REGION Network 61: PHMI Servo Enable CMs
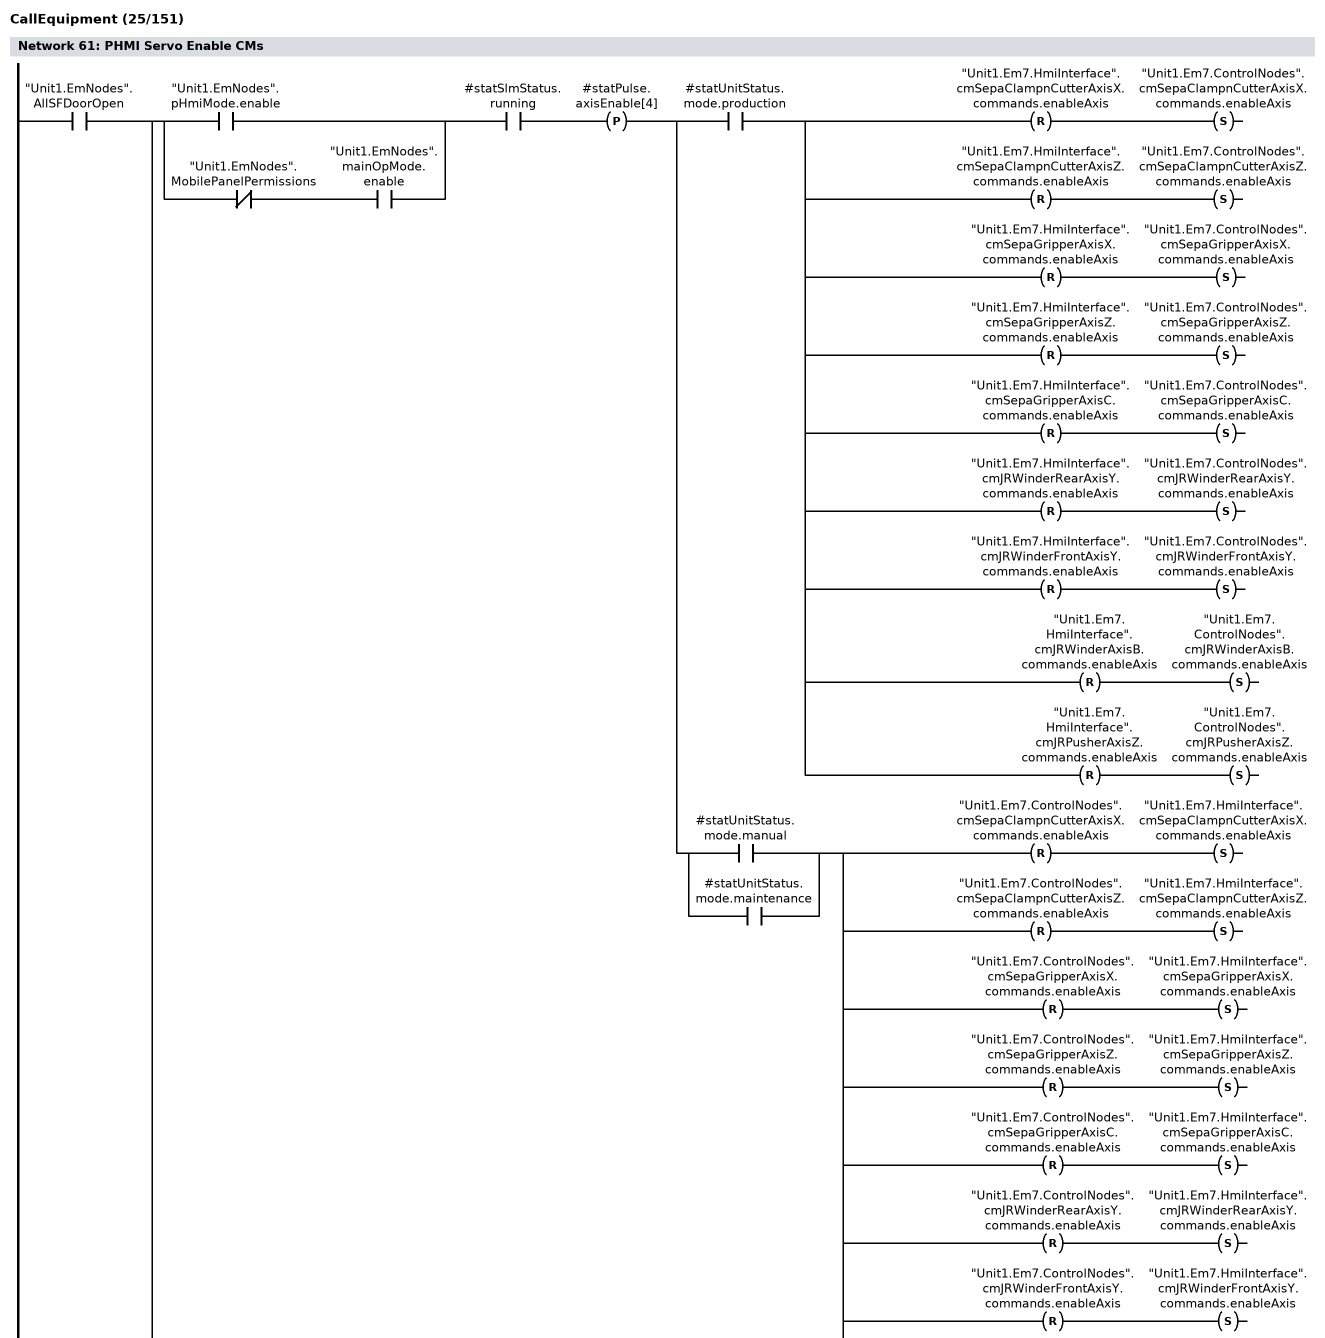
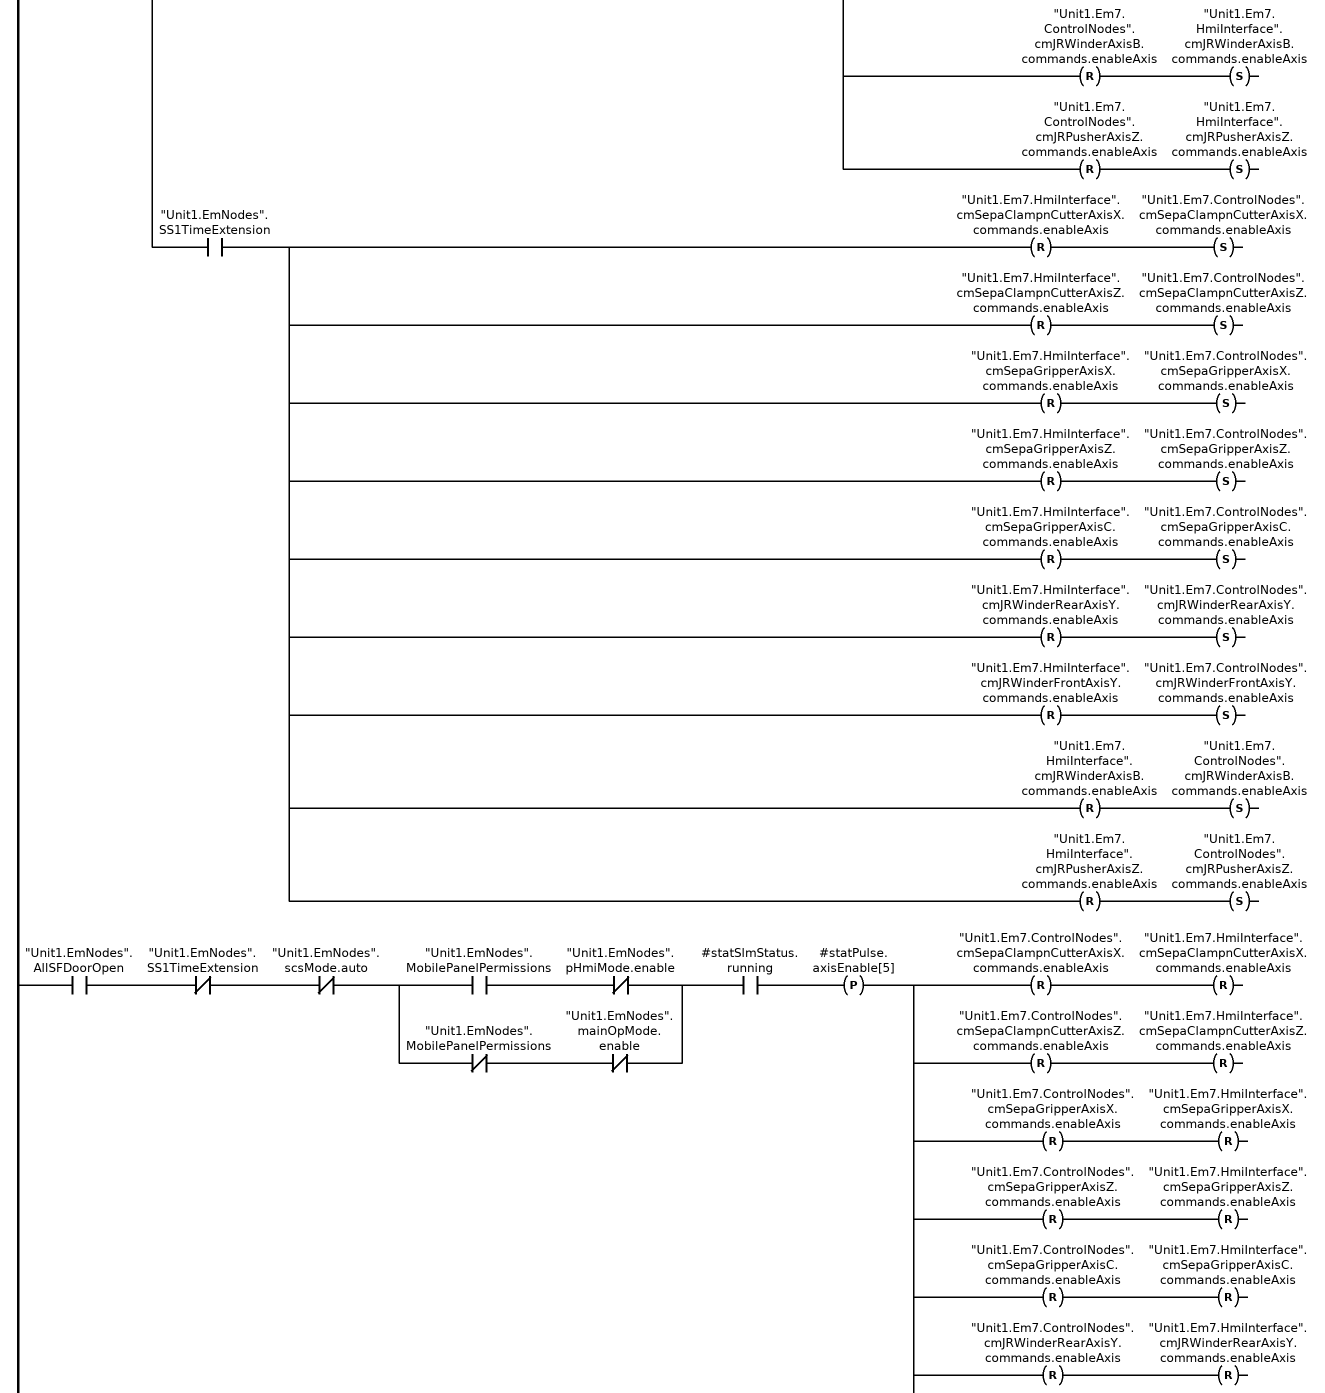
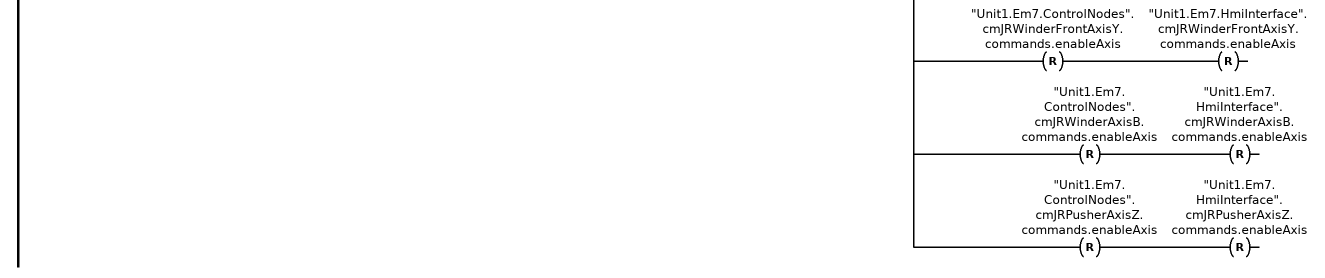
   RUNG wire#powerrail
      Contact( "Unit1.EmNodes".AllSFDoorOpen )
      wire#w1
      Contact( "Unit1.EmNodes".pHmiMode.enable )
      wire#w2
      Contact( #statSlmStatus.running )
      P_Trig( #statPulse.axisEnable[4] )
      wire#w3
      Contact( #statUnitStatus.mode.production )
      wire#w4
      R_Coil( "Unit1.Em7.HmiInterface".cmSepaClampnCutterAxisX.commands.enableAxis )
      S_Coil( "Unit1.Em7.ControlNodes".cmSepaClampnCutterAxisX.commands.enableAxis )
   END_RUNG
   RUNG wire#w1
      I_Contact( "Unit1.EmNodes".MobilePanelPermissions )
      Contact( "Unit1.EmNodes".mainOpMode.enable )
   END_RUNG wire#w2
   RUNG wire#w4
      R_Coil( "Unit1.Em7.HmiInterface".cmSepaClampnCutterAxisZ.commands.enableAxis )
      S_Coil( "Unit1.Em7.ControlNodes".cmSepaClampnCutterAxisZ.commands.enableAxis )
   END_RUNG
   RUNG wire#w4
      R_Coil( "Unit1.Em7.HmiInterface".cmSepaGripperAxisX.commands.enableAxis )
      S_Coil( "Unit1.Em7.ControlNodes".cmSepaGripperAxisX.commands.enableAxis )
   END_RUNG
   RUNG wire#w4
      R_Coil( "Unit1.Em7.HmiInterface".cmSepaGripperAxisZ.commands.enableAxis )
      S_Coil( "Unit1.Em7.ControlNodes".cmSepaGripperAxisZ.commands.enableAxis )
   END_RUNG
   RUNG wire#w4
      R_Coil( "Unit1.Em7.HmiInterface".cmSepaGripperAxisC.commands.enableAxis )
      S_Coil( "Unit1.Em7.ControlNodes".cmSepaGripperAxisC.commands.enableAxis )
   END_RUNG
   RUNG wire#w4
      R_Coil( "Unit1.Em7.HmiInterface".cmJRWinderRearAxisY.commands.enableAxis )
      S_Coil( "Unit1.Em7.ControlNodes".cmJRWinderRearAxisY.commands.enableAxis )
   END_RUNG
   RUNG wire#w4
      R_Coil( "Unit1.Em7.HmiInterface".cmJRWinderFrontAxisY.commands.enableAxis )
      S_Coil( "Unit1.Em7.ControlNodes".cmJRWinderFrontAxisY.commands.enableAxis )
   END_RUNG
   RUNG wire#w4
      R_Coil( "Unit1.Em7.HmiInterface".cmJRWinderAxisB.commands.enableAxis )
      S_Coil( "Unit1.Em7.ControlNodes".cmJRWinderAxisB.commands.enableAxis )
   END_RUNG
   RUNG wire#w4
      R_Coil( "Unit1.Em7.HmiInterface".cmJRPusherAxisZ.commands.enableAxis )
      S_Coil( "Unit1.Em7.ControlNodes".cmJRPusherAxisZ.commands.enableAxis )
   END_RUNG
   RUNG wire#w3
      Contact( #statUnitStatus.mode.manual )
      wire#w5
      R_Coil( "Unit1.Em7.ControlNodes".cmSepaClampnCutterAxisX.commands.enableAxis )
      S_Coil( "Unit1.Em7.HmiInterface".cmSepaClampnCutterAxisX.commands.enableAxis )
   END_RUNG
   RUNG wire#w3
      Contact( #statUnitStatus.mode.maintenance )
   END_RUNG wire#w5
   RUNG wire#w5
      R_Coil( "Unit1.Em7.ControlNodes".cmSepaClampnCutterAxisZ.commands.enableAxis )
      S_Coil( "Unit1.Em7.HmiInterface".cmSepaClampnCutterAxisZ.commands.enableAxis )
   END_RUNG
   RUNG wire#w5
      R_Coil( "Unit1.Em7.ControlNodes".cmSepaGripperAxisX.commands.enableAxis )
      S_Coil( "Unit1.Em7.HmiInterface".cmSepaGripperAxisX.commands.enableAxis )
   END_RUNG
   RUNG wire#w5
      R_Coil( "Unit1.Em7.ControlNodes".cmSepaGripperAxisZ.commands.enableAxis )
      S_Coil( "Unit1.Em7.HmiInterface".cmSepaGripperAxisZ.commands.enableAxis )
   END_RUNG
   RUNG wire#w5
      R_Coil( "Unit1.Em7.ControlNodes".cmSepaGripperAxisC.commands.enableAxis )
      S_Coil( "Unit1.Em7.HmiInterface".cmSepaGripperAxisC.commands.enableAxis )
   END_RUNG
   RUNG wire#w5
      R_Coil( "Unit1.Em7.ControlNodes".cmJRWinderRearAxisY.commands.enableAxis )
      S_Coil( "Unit1.Em7.HmiInterface".cmJRWinderRearAxisY.commands.enableAxis )
   END_RUNG
   RUNG wire#w5
      R_Coil( "Unit1.Em7.ControlNodes".cmJRWinderFrontAxisY.commands.enableAxis )
      S_Coil( "Unit1.Em7.HmiInterface".cmJRWinderFrontAxisY.commands.enableAxis )
   END_RUNG
   RUNG wire#w5
      R_Coil( "Unit1.Em7.ControlNodes".cmJRWinderAxisB.commands.enableAxis )
      S_Coil( "Unit1.Em7.HmiInterface".cmJRWinderAxisB.commands.enableAxis )
   END_RUNG
   RUNG wire#w5
      R_Coil( "Unit1.Em7.ControlNodes".cmJRPusherAxisZ.commands.enableAxis )
      S_Coil( "Unit1.Em7.HmiInterface".cmJRPusherAxisZ.commands.enableAxis )
   END_RUNG
   RUNG wire#w1
      Contact( "Unit1.EmNodes".SS1TimeExtension )
      wire#w6
      R_Coil( "Unit1.Em7.HmiInterface".cmSepaClampnCutterAxisX.commands.enableAxis )
      S_Coil( "Unit1.Em7.ControlNodes".cmSepaClampnCutterAxisX.commands.enableAxis )
   END_RUNG
   RUNG wire#w6
      R_Coil( "Unit1.Em7.HmiInterface".cmSepaClampnCutterAxisZ.commands.enableAxis )
      S_Coil( "Unit1.Em7.ControlNodes".cmSepaClampnCutterAxisZ.commands.enableAxis )
   END_RUNG
   RUNG wire#w6
      R_Coil( "Unit1.Em7.HmiInterface".cmSepaGripperAxisX.commands.enableAxis )
      S_Coil( "Unit1.Em7.ControlNodes".cmSepaGripperAxisX.commands.enableAxis )
   END_RUNG
   RUNG wire#w6
      R_Coil( "Unit1.Em7.HmiInterface".cmSepaGripperAxisZ.commands.enableAxis )
      S_Coil( "Unit1.Em7.ControlNodes".cmSepaGripperAxisZ.commands.enableAxis )
   END_RUNG
   RUNG wire#w6
      R_Coil( "Unit1.Em7.HmiInterface".cmSepaGripperAxisC.commands.enableAxis )
      S_Coil( "Unit1.Em7.ControlNodes".cmSepaGripperAxisC.commands.enableAxis )
   END_RUNG
   RUNG wire#w6
      R_Coil( "Unit1.Em7.HmiInterface".cmJRWinderRearAxisY.commands.enableAxis )
      S_Coil( "Unit1.Em7.ControlNodes".cmJRWinderRearAxisY.commands.enableAxis )
   END_RUNG
   RUNG wire#w6
      R_Coil( "Unit1.Em7.HmiInterface".cmJRWinderFrontAxisY.commands.enableAxis )
      S_Coil( "Unit1.Em7.ControlNodes".cmJRWinderFrontAxisY.commands.enableAxis )
   END_RUNG
   RUNG wire#w6
      R_Coil( "Unit1.Em7.HmiInterface".cmJRWinderAxisB.commands.enableAxis )
      S_Coil( "Unit1.Em7.ControlNodes".cmJRWinderAxisB.commands.enableAxis )
   END_RUNG
   RUNG wire#w6
      R_Coil( "Unit1.Em7.HmiInterface".cmJRPusherAxisZ.commands.enableAxis )
      S_Coil( "Unit1.Em7.ControlNodes".cmJRPusherAxisZ.commands.enableAxis )
   END_RUNG
   RUNG wire#powerrail
      Contact( "Unit1.EmNodes".AllSFDoorOpen )
      I_Contact( "Unit1.EmNodes".SS1TimeExtension )
      I_Contact( "Unit1.EmNodes".scsMode.auto )
      wire#w7
      Contact( "Unit1.EmNodes".MobilePanelPermissions )
      I_Contact( "Unit1.EmNodes".pHmiMode.enable )
      wire#w8
      Contact( #statSlmStatus.running )
      P_Trig( #statPulse.axisEnable[5] )
      wire#w9
      R_Coil( "Unit1.Em7.ControlNodes".cmSepaClampnCutterAxisX.commands.enableAxis )
      R_Coil( "Unit1.Em7.HmiInterface".cmSepaClampnCutterAxisX.commands.enableAxis )
   END_RUNG
   RUNG wire#w7
      I_Contact( "Unit1.EmNodes".MobilePanelPermissions )
      I_Contact( "Unit1.EmNodes".mainOpMode.enable )
   END_RUNG wire#w8
   RUNG wire#w9
      R_Coil( "Unit1.Em7.ControlNodes".cmSepaClampnCutterAxisZ.commands.enableAxis )
      R_Coil( "Unit1.Em7.HmiInterface".cmSepaClampnCutterAxisZ.commands.enableAxis )
   END_RUNG
   RUNG wire#w9
      R_Coil( "Unit1.Em7.ControlNodes".cmSepaGripperAxisX.commands.enableAxis )
      R_Coil( "Unit1.Em7.HmiInterface".cmSepaGripperAxisX.commands.enableAxis )
   END_RUNG
   RUNG wire#w9
      R_Coil( "Unit1.Em7.ControlNodes".cmSepaGripperAxisZ.commands.enableAxis )
      R_Coil( "Unit1.Em7.HmiInterface".cmSepaGripperAxisZ.commands.enableAxis )
   END_RUNG
   RUNG wire#w9
      R_Coil( "Unit1.Em7.ControlNodes".cmSepaGripperAxisC.commands.enableAxis )
      R_Coil( "Unit1.Em7.HmiInterface".cmSepaGripperAxisC.commands.enableAxis )
   END_RUNG
   RUNG wire#w9
      R_Coil( "Unit1.Em7.ControlNodes".cmJRWinderRearAxisY.commands.enableAxis )
      R_Coil( "Unit1.Em7.HmiInterface".cmJRWinderRearAxisY.commands.enableAxis )
   END_RUNG
   RUNG wire#w9
      R_Coil( "Unit1.Em7.ControlNodes".cmJRWinderFrontAxisY.commands.enableAxis )
      R_Coil( "Unit1.Em7.HmiInterface".cmJRWinderFrontAxisY.commands.enableAxis )
   END_RUNG
   RUNG wire#w9
      R_Coil( "Unit1.Em7.ControlNodes".cmJRWinderAxisB.commands.enableAxis )
      R_Coil( "Unit1.Em7.HmiInterface".cmJRWinderAxisB.commands.enableAxis )
   END_RUNG
   RUNG wire#w9
      R_Coil( "Unit1.Em7.ControlNodes".cmJRPusherAxisZ.commands.enableAxis )
      R_Coil( "Unit1.Em7.HmiInterface".cmJRPusherAxisZ.commands.enableAxis )
   END_RUNG
   // the same network as SCL:
   #_w1 := "Unit1.EmNodes".AllSFDoorOpen AND ("Unit1.EmNodes".pHmiMode.enable OR (NOT "Unit1.EmNodes".MobilePanelPermissions AND "Unit1.EmNodes".mainOpMode.enable)) AND #statSlmStatus.running;
   #_w2 := #_w1 AND NOT #statPulse.axisEnable[4];   // rising edge
   #statPulse.axisEnable[4] := #_w1;
   IF #_w2 AND #statUnitStatus.mode.production THEN
       "Unit1.Em7.HmiInterface".cmSepaClampnCutterAxisX.commands.enableAxis := FALSE;
       "Unit1.Em7.ControlNodes".cmSepaClampnCutterAxisX.commands.enableAxis := TRUE;
       "Unit1.Em7.HmiInterface".cmSepaClampnCutterAxisZ.commands.enableAxis := FALSE;
       "Unit1.Em7.ControlNodes".cmSepaClampnCutterAxisZ.commands.enableAxis := TRUE;
       "Unit1.Em7.HmiInterface".cmSepaGripperAxisX.commands.enableAxis := FALSE;
       "Unit1.Em7.ControlNodes".cmSepaGripperAxisX.commands.enableAxis := TRUE;
       "Unit1.Em7.HmiInterface".cmSepaGripperAxisZ.commands.enableAxis := FALSE;
       "Unit1.Em7.ControlNodes".cmSepaGripperAxisZ.commands.enableAxis := TRUE;
       "Unit1.Em7.HmiInterface".cmSepaGripperAxisC.commands.enableAxis := FALSE;
       "Unit1.Em7.ControlNodes".cmSepaGripperAxisC.commands.enableAxis := TRUE;
       "Unit1.Em7.HmiInterface".cmJRWinderRearAxisY.commands.enableAxis := FALSE;
       "Unit1.Em7.ControlNodes".cmJRWinderRearAxisY.commands.enableAxis := TRUE;
       "Unit1.Em7.HmiInterface".cmJRWinderFrontAxisY.commands.enableAxis := FALSE;
       "Unit1.Em7.ControlNodes".cmJRWinderFrontAxisY.commands.enableAxis := TRUE;
       "Unit1.Em7.HmiInterface".cmJRWinderAxisB.commands.enableAxis := FALSE;
       "Unit1.Em7.ControlNodes".cmJRWinderAxisB.commands.enableAxis := TRUE;
       "Unit1.Em7.HmiInterface".cmJRPusherAxisZ.commands.enableAxis := FALSE;
       "Unit1.Em7.ControlNodes".cmJRPusherAxisZ.commands.enableAxis := TRUE;
   END_IF;
   IF #_w2 AND (#statUnitStatus.mode.manual OR #statUnitStatus.mode.maintenance) THEN
       "Unit1.Em7.ControlNodes".cmSepaClampnCutterAxisX.commands.enableAxis := FALSE;
       "Unit1.Em7.HmiInterface".cmSepaClampnCutterAxisX.commands.enableAxis := TRUE;
       "Unit1.Em7.ControlNodes".cmSepaClampnCutterAxisZ.commands.enableAxis := FALSE;
       "Unit1.Em7.HmiInterface".cmSepaClampnCutterAxisZ.commands.enableAxis := TRUE;
       "Unit1.Em7.ControlNodes".cmSepaGripperAxisX.commands.enableAxis := FALSE;
       "Unit1.Em7.HmiInterface".cmSepaGripperAxisX.commands.enableAxis := TRUE;
       "Unit1.Em7.ControlNodes".cmSepaGripperAxisZ.commands.enableAxis := FALSE;
       "Unit1.Em7.HmiInterface".cmSepaGripperAxisZ.commands.enableAxis := TRUE;
       "Unit1.Em7.ControlNodes".cmSepaGripperAxisC.commands.enableAxis := FALSE;
       "Unit1.Em7.HmiInterface".cmSepaGripperAxisC.commands.enableAxis := TRUE;
       "Unit1.Em7.ControlNodes".cmJRWinderRearAxisY.commands.enableAxis := FALSE;
       "Unit1.Em7.HmiInterface".cmJRWinderRearAxisY.commands.enableAxis := TRUE;
       "Unit1.Em7.ControlNodes".cmJRWinderFrontAxisY.commands.enableAxis := FALSE;
       "Unit1.Em7.HmiInterface".cmJRWinderFrontAxisY.commands.enableAxis := TRUE;
       "Unit1.Em7.ControlNodes".cmJRWinderAxisB.commands.enableAxis := FALSE;
       "Unit1.Em7.HmiInterface".cmJRWinderAxisB.commands.enableAxis := TRUE;
       "Unit1.Em7.ControlNodes".cmJRPusherAxisZ.commands.enableAxis := FALSE;
       "Unit1.Em7.HmiInterface".cmJRPusherAxisZ.commands.enableAxis := TRUE;
   END_IF;
   IF "Unit1.EmNodes".AllSFDoorOpen AND "Unit1.EmNodes".SS1TimeExtension THEN
       "Unit1.Em7.HmiInterface".cmSepaClampnCutterAxisX.commands.enableAxis := FALSE;
       "Unit1.Em7.ControlNodes".cmSepaClampnCutterAxisX.commands.enableAxis := TRUE;
       "Unit1.Em7.HmiInterface".cmSepaClampnCutterAxisZ.commands.enableAxis := FALSE;
       "Unit1.Em7.ControlNodes".cmSepaClampnCutterAxisZ.commands.enableAxis := TRUE;
       "Unit1.Em7.HmiInterface".cmSepaGripperAxisX.commands.enableAxis := FALSE;
       "Unit1.Em7.ControlNodes".cmSepaGripperAxisX.commands.enableAxis := TRUE;
       "Unit1.Em7.HmiInterface".cmSepaGripperAxisZ.commands.enableAxis := FALSE;
       "Unit1.Em7.ControlNodes".cmSepaGripperAxisZ.commands.enableAxis := TRUE;
       "Unit1.Em7.HmiInterface".cmSepaGripperAxisC.commands.enableAxis := FALSE;
       "Unit1.Em7.ControlNodes".cmSepaGripperAxisC.commands.enableAxis := TRUE;
       "Unit1.Em7.HmiInterface".cmJRWinderRearAxisY.commands.enableAxis := FALSE;
       "Unit1.Em7.ControlNodes".cmJRWinderRearAxisY.commands.enableAxis := TRUE;
       "Unit1.Em7.HmiInterface".cmJRWinderFrontAxisY.commands.enableAxis := FALSE;
       "Unit1.Em7.ControlNodes".cmJRWinderFrontAxisY.commands.enableAxis := TRUE;
       "Unit1.Em7.HmiInterface".cmJRWinderAxisB.commands.enableAxis := FALSE;
       "Unit1.Em7.ControlNodes".cmJRWinderAxisB.commands.enableAxis := TRUE;
       "Unit1.Em7.HmiInterface".cmJRPusherAxisZ.commands.enableAxis := FALSE;
       "Unit1.Em7.ControlNodes".cmJRPusherAxisZ.commands.enableAxis := TRUE;
   END_IF;
   #_w3 := "Unit1.EmNodes".AllSFDoorOpen AND NOT "Unit1.EmNodes".SS1TimeExtension AND NOT "Unit1.EmNodes".scsMode.auto AND (("Unit1.EmNodes".MobilePanelPermissions AND NOT "Unit1.EmNodes".pHmiMode.enable) OR (NOT "Unit1.EmNodes".MobilePanelPermissions AND NOT "Unit1.EmNodes".mainOpMode.enable)) AND #statSlmStatus.running;
   #_w4 := #_w3 AND NOT #statPulse.axisEnable[5];   // rising edge
   #statPulse.axisEnable[5] := #_w3;
   IF #_w4 THEN
       "Unit1.Em7.ControlNodes".cmSepaClampnCutterAxisX.commands.enableAxis := FALSE;
       "Unit1.Em7.HmiInterface".cmSepaClampnCutterAxisX.commands.enableAxis := FALSE;
       "Unit1.Em7.ControlNodes".cmSepaClampnCutterAxisZ.commands.enableAxis := FALSE;
       "Unit1.Em7.HmiInterface".cmSepaClampnCutterAxisZ.commands.enableAxis := FALSE;
       "Unit1.Em7.ControlNodes".cmSepaGripperAxisX.commands.enableAxis := FALSE;
       "Unit1.Em7.HmiInterface".cmSepaGripperAxisX.commands.enableAxis := FALSE;
       "Unit1.Em7.ControlNodes".cmSepaGripperAxisZ.commands.enableAxis := FALSE;
       "Unit1.Em7.HmiInterface".cmSepaGripperAxisZ.commands.enableAxis := FALSE;
       "Unit1.Em7.ControlNodes".cmSepaGripperAxisC.commands.enableAxis := FALSE;
       "Unit1.Em7.HmiInterface".cmSepaGripperAxisC.commands.enableAxis := FALSE;
       "Unit1.Em7.ControlNodes".cmJRWinderRearAxisY.commands.enableAxis := FALSE;
       "Unit1.Em7.HmiInterface".cmJRWinderRearAxisY.commands.enableAxis := FALSE;
       "Unit1.Em7.ControlNodes".cmJRWinderFrontAxisY.commands.enableAxis := FALSE;
       "Unit1.Em7.HmiInterface".cmJRWinderFrontAxisY.commands.enableAxis := FALSE;
       "Unit1.Em7.ControlNodes".cmJRWinderAxisB.commands.enableAxis := FALSE;
       "Unit1.Em7.HmiInterface".cmJRWinderAxisB.commands.enableAxis := FALSE;
       "Unit1.Em7.ControlNodes".cmJRPusherAxisZ.commands.enableAxis := FALSE;
       "Unit1.Em7.HmiInterface".cmJRPusherAxisZ.commands.enableAxis := FALSE;
   END_IF;
END_REGION

REGION Network 62: Disable All CMs
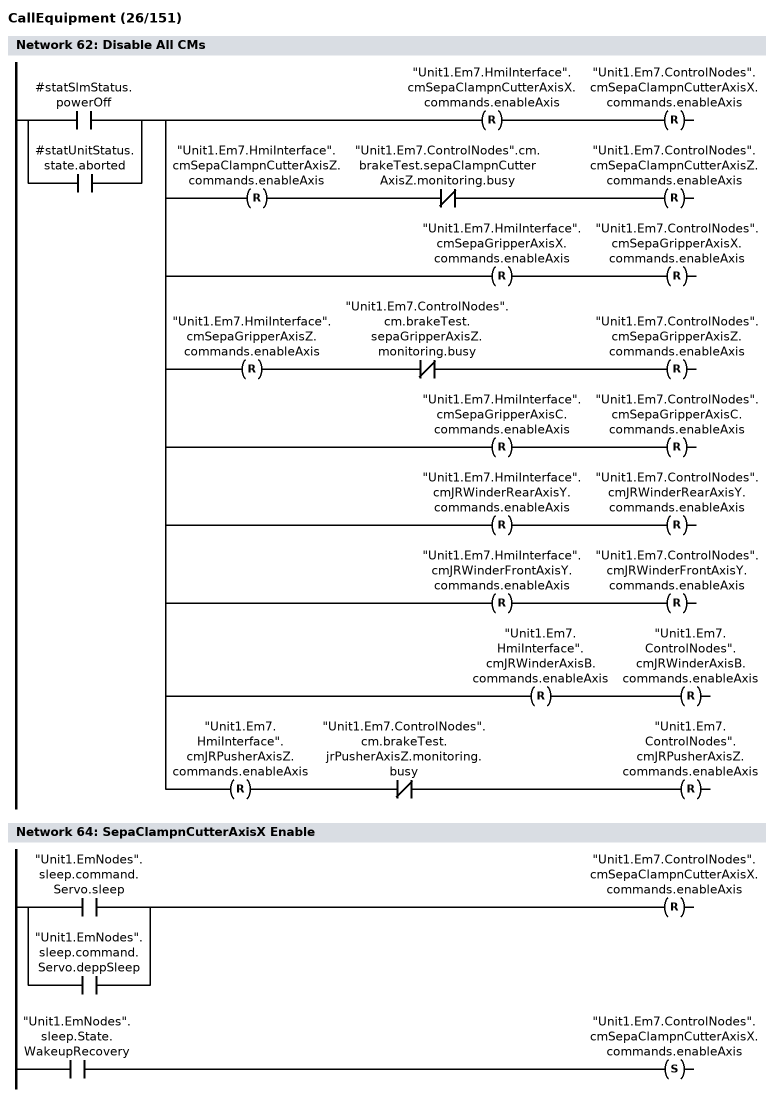
   RUNG wire#powerrail
      Contact( #statSlmStatus.powerOff )
      wire#w1
      R_Coil( "Unit1.Em7.HmiInterface".cmSepaClampnCutterAxisX.commands.enableAxis )
      R_Coil( "Unit1.Em7.ControlNodes".cmSepaClampnCutterAxisX.commands.enableAxis )
   END_RUNG
   RUNG wire#powerrail
      Contact( #statUnitStatus.state.aborted )
   END_RUNG wire#w1
   RUNG wire#w1
      R_Coil( "Unit1.Em7.HmiInterface".cmSepaClampnCutterAxisZ.commands.enableAxis )
      I_Contact( "Unit1.Em7.ControlNodes".cm.brakeTest.sepaClampnCutterAxisZ.monitoring.busy )
      R_Coil( "Unit1.Em7.ControlNodes".cmSepaClampnCutterAxisZ.commands.enableAxis )
   END_RUNG
   RUNG wire#w1
      R_Coil( "Unit1.Em7.HmiInterface".cmSepaGripperAxisX.commands.enableAxis )
      R_Coil( "Unit1.Em7.ControlNodes".cmSepaGripperAxisX.commands.enableAxis )
   END_RUNG
   RUNG wire#w1
      R_Coil( "Unit1.Em7.HmiInterface".cmSepaGripperAxisZ.commands.enableAxis )
      I_Contact( "Unit1.Em7.ControlNodes".cm.brakeTest.sepaGripperAxisZ.monitoring.busy )
      R_Coil( "Unit1.Em7.ControlNodes".cmSepaGripperAxisZ.commands.enableAxis )
   END_RUNG
   RUNG wire#w1
      R_Coil( "Unit1.Em7.HmiInterface".cmSepaGripperAxisC.commands.enableAxis )
      R_Coil( "Unit1.Em7.ControlNodes".cmSepaGripperAxisC.commands.enableAxis )
   END_RUNG
   RUNG wire#w1
      R_Coil( "Unit1.Em7.HmiInterface".cmJRWinderRearAxisY.commands.enableAxis )
      R_Coil( "Unit1.Em7.ControlNodes".cmJRWinderRearAxisY.commands.enableAxis )
   END_RUNG
   RUNG wire#w1
      R_Coil( "Unit1.Em7.HmiInterface".cmJRWinderFrontAxisY.commands.enableAxis )
      R_Coil( "Unit1.Em7.ControlNodes".cmJRWinderFrontAxisY.commands.enableAxis )
   END_RUNG
   RUNG wire#w1
      R_Coil( "Unit1.Em7.HmiInterface".cmJRWinderAxisB.commands.enableAxis )
      R_Coil( "Unit1.Em7.ControlNodes".cmJRWinderAxisB.commands.enableAxis )
   END_RUNG
   RUNG wire#w1
      R_Coil( "Unit1.Em7.HmiInterface".cmJRPusherAxisZ.commands.enableAxis )
      I_Contact( "Unit1.Em7.ControlNodes".cm.brakeTest.jrPusherAxisZ.monitoring.busy )
      R_Coil( "Unit1.Em7.ControlNodes".cmJRPusherAxisZ.commands.enableAxis )
   END_RUNG
   // the same network as SCL:
   #_w1 := #statSlmStatus.powerOff OR #statUnitStatus.state.aborted;
   IF #_w1 THEN
       "Unit1.Em7.HmiInterface".cmSepaClampnCutterAxisX.commands.enableAxis := FALSE;
       "Unit1.Em7.ControlNodes".cmSepaClampnCutterAxisX.commands.enableAxis := FALSE;
       "Unit1.Em7.HmiInterface".cmSepaClampnCutterAxisZ.commands.enableAxis := FALSE;
   END_IF;
   IF #_w1 AND NOT "Unit1.Em7.ControlNodes".cm.brakeTest.sepaClampnCutterAxisZ.monitoring.busy THEN
       "Unit1.Em7.ControlNodes".cmSepaClampnCutterAxisZ.commands.enableAxis := FALSE;
   END_IF;
   IF #_w1 THEN
       "Unit1.Em7.HmiInterface".cmSepaGripperAxisX.commands.enableAxis := FALSE;
       "Unit1.Em7.ControlNodes".cmSepaGripperAxisX.commands.enableAxis := FALSE;
       "Unit1.Em7.HmiInterface".cmSepaGripperAxisZ.commands.enableAxis := FALSE;
   END_IF;
   IF #_w1 AND NOT "Unit1.Em7.ControlNodes".cm.brakeTest.sepaGripperAxisZ.monitoring.busy THEN
       "Unit1.Em7.ControlNodes".cmSepaGripperAxisZ.commands.enableAxis := FALSE;
   END_IF;
   IF #_w1 THEN
       "Unit1.Em7.HmiInterface".cmSepaGripperAxisC.commands.enableAxis := FALSE;
       "Unit1.Em7.ControlNodes".cmSepaGripperAxisC.commands.enableAxis := FALSE;
       "Unit1.Em7.HmiInterface".cmJRWinderRearAxisY.commands.enableAxis := FALSE;
       "Unit1.Em7.ControlNodes".cmJRWinderRearAxisY.commands.enableAxis := FALSE;
       "Unit1.Em7.HmiInterface".cmJRWinderFrontAxisY.commands.enableAxis := FALSE;
       "Unit1.Em7.ControlNodes".cmJRWinderFrontAxisY.commands.enableAxis := FALSE;
       "Unit1.Em7.HmiInterface".cmJRWinderAxisB.commands.enableAxis := FALSE;
       "Unit1.Em7.ControlNodes".cmJRWinderAxisB.commands.enableAxis := FALSE;
       "Unit1.Em7.HmiInterface".cmJRPusherAxisZ.commands.enableAxis := FALSE;
   END_IF;
   IF #_w1 AND NOT "Unit1.Em7.ControlNodes".cm.brakeTest.jrPusherAxisZ.monitoring.busy THEN
       "Unit1.Em7.ControlNodes".cmJRPusherAxisZ.commands.enableAxis := FALSE;
   END_IF;
END_REGION

REGION Network 64: SepaClampnCutterAxisX Enable
   RUNG wire#powerrail
      Contact( "Unit1.EmNodes".sleep.command.Servo.sleep )
      wire#w1
      R_Coil( "Unit1.Em7.ControlNodes".cmSepaClampnCutterAxisX.commands.enableAxis )
   END_RUNG
   RUNG wire#powerrail
      Contact( "Unit1.EmNodes".sleep.command.Servo.deppSleep )
   END_RUNG wire#w1
   RUNG wire#powerrail
      Contact( "Unit1.EmNodes".sleep.State.WakeupRecovery )
      S_Coil( "Unit1.Em7.ControlNodes".cmSepaClampnCutterAxisX.commands.enableAxis )
   END_RUNG
   // the same network as SCL:
   IF "Unit1.EmNodes".sleep.command.Servo.sleep OR "Unit1.EmNodes".sleep.command.Servo.deppSleep THEN
       "Unit1.Em7.ControlNodes".cmSepaClampnCutterAxisX.commands.enableAxis := FALSE;
   END_IF;
   IF "Unit1.EmNodes".sleep.State.WakeupRecovery THEN
       "Unit1.Em7.ControlNodes".cmSepaClampnCutterAxisX.commands.enableAxis := TRUE;
   END_IF;
END_REGION

REGION Network 65: CmSepaClampnCutterAxisX Position Absolute Home
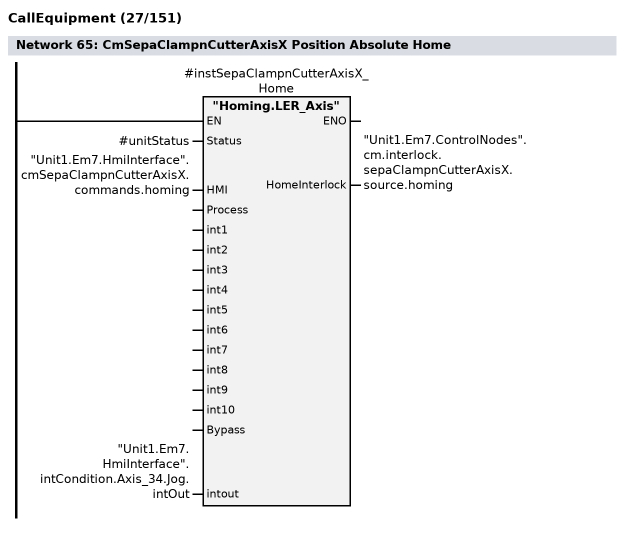
   RUNG wire#powerrail
      #instSepaClampnCutterAxisX_Home(Status := #unitStatus, HMI := "Unit1.Em7.HmiInterface".cmSepaClampnCutterAxisX.commands.homing, Process :=, int1 :=, int2 :=, int3 :=, int4 :=, int5 :=, int6 :=, int7 :=, int8 :=, int9 :=, int10 :=, Bypass :=, intout := "Unit1.Em7.HmiInterface".intCondition.Axis_34.Jog.intOut, HomeInterlock => "Unit1.Em7.ControlNodes".cm.interlock.sepaClampnCutterAxisX.source.homing)
   END_RUNG
   // the same network as SCL:
   #instSepaClampnCutterAxisX_Home(Status := #unitStatus,   // "Homing.LER_Axis"
                           HMI := "Unit1.Em7.HmiInterface".cmSepaClampnCutterAxisX.commands.homing,
                           intout := "Unit1.Em7.HmiInterface".intCondition.Axis_34.Jog.intOut,
                           HomeInterlock => "Unit1.Em7.ControlNodes".cm.interlock.sepaClampnCutterAxisX.source.homing);
END_REGION

REGION Network 66: CmSepaClampnCutterAxisX Position Absolute Jog
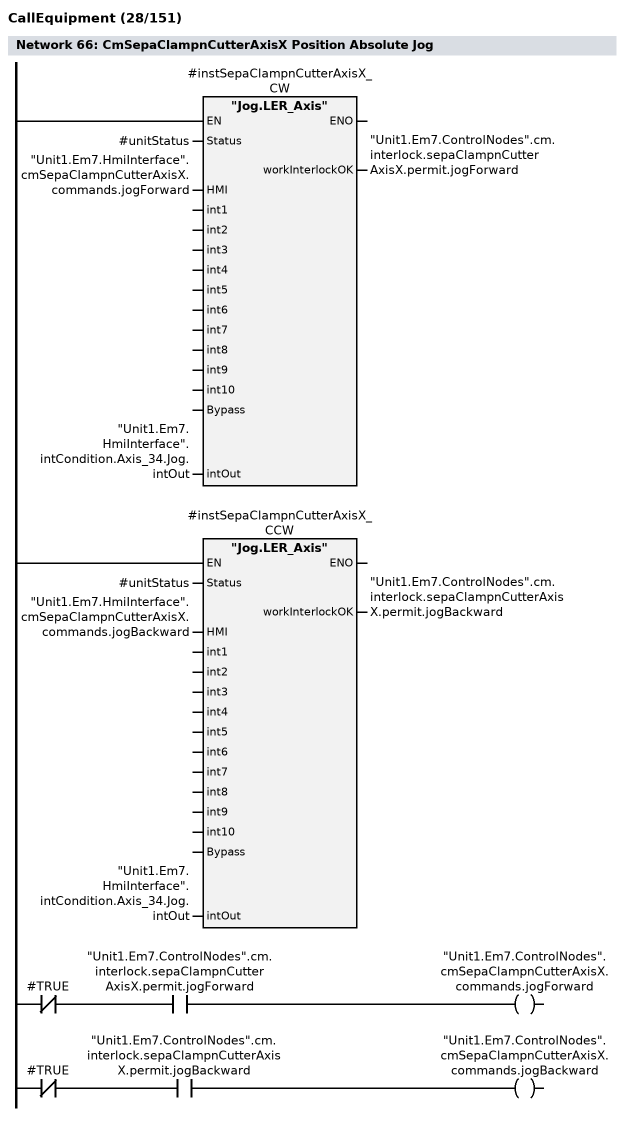
   RUNG wire#powerrail
      #instSepaClampnCutterAxisX_CW(Status := #unitStatus, HMI := "Unit1.Em7.HmiInterface".cmSepaClampnCutterAxisX.commands.jogForward, int1 :=, int2 :=, int3 :=, int4 :=, int5 :=, int6 :=, int7 :=, int8 :=, int9 :=, int10 :=, Bypass :=, intOut := "Unit1.Em7.HmiInterface".intCondition.Axis_34.Jog.intOut, workInterlockOK => "Unit1.Em7.ControlNodes".cm.interlock.sepaClampnCutterAxisX.permit.jogForward)
   END_RUNG
   RUNG wire#powerrail
      #instSepaClampnCutterAxisX_CCW(Status := #unitStatus, HMI := "Unit1.Em7.HmiInterface".cmSepaClampnCutterAxisX.commands.jogBackward, int1 :=, int2 :=, int3 :=, int4 :=, int5 :=, int6 :=, int7 :=, int8 :=, int9 :=, int10 :=, Bypass :=, intOut := "Unit1.Em7.HmiInterface".intCondition.Axis_34.Jog.intOut, workInterlockOK => "Unit1.Em7.ControlNodes".cm.interlock.sepaClampnCutterAxisX.permit.jogBackward)
   END_RUNG
   RUNG wire#powerrail
      I_Contact( #TRUE )
      Contact( "Unit1.Em7.ControlNodes".cm.interlock.sepaClampnCutterAxisX.permit.jogForward )
      Coil( "Unit1.Em7.ControlNodes".cmSepaClampnCutterAxisX.commands.jogForward )
   END_RUNG
   RUNG wire#powerrail
      I_Contact( #TRUE )
      Contact( "Unit1.Em7.ControlNodes".cm.interlock.sepaClampnCutterAxisX.permit.jogBackward )
      Coil( "Unit1.Em7.ControlNodes".cmSepaClampnCutterAxisX.commands.jogBackward )
   END_RUNG
   // the same network as SCL:
   #instSepaClampnCutterAxisX_CW(Status := #unitStatus,   // "Jog.LER_Axis"
                           HMI := "Unit1.Em7.HmiInterface".cmSepaClampnCutterAxisX.commands.jogForward,
                           intOut := "Unit1.Em7.HmiInterface".intCondition.Axis_34.Jog.intOut,
                           workInterlockOK => "Unit1.Em7.ControlNodes".cm.interlock.sepaClampnCutterAxisX.permit.jogForward);
   #instSepaClampnCutterAxisX_CCW(Status := #unitStatus,   // "Jog.LER_Axis"
                           HMI := "Unit1.Em7.HmiInterface".cmSepaClampnCutterAxisX.commands.jogBackward,
                           intOut := "Unit1.Em7.HmiInterface".intCondition.Axis_34.Jog.intOut,
                           workInterlockOK => "Unit1.Em7.ControlNodes".cm.interlock.sepaClampnCutterAxisX.permit.jogBackward);
   "Unit1.Em7.ControlNodes".cmSepaClampnCutterAxisX.commands.jogForward := NOT #TRUE AND "Unit1.Em7.ControlNodes".cm.interlock.sepaClampnCutterAxisX.permit.jogForward;
   "Unit1.Em7.ControlNodes".cmSepaClampnCutterAxisX.commands.jogBackward := NOT #TRUE AND "Unit1.Em7.ControlNodes".cm.interlock.sepaClampnCutterAxisX.permit.jogBackward;
END_REGION

REGION Network 67: CmSepaClampnCutterAxisX Position Absolute Position0
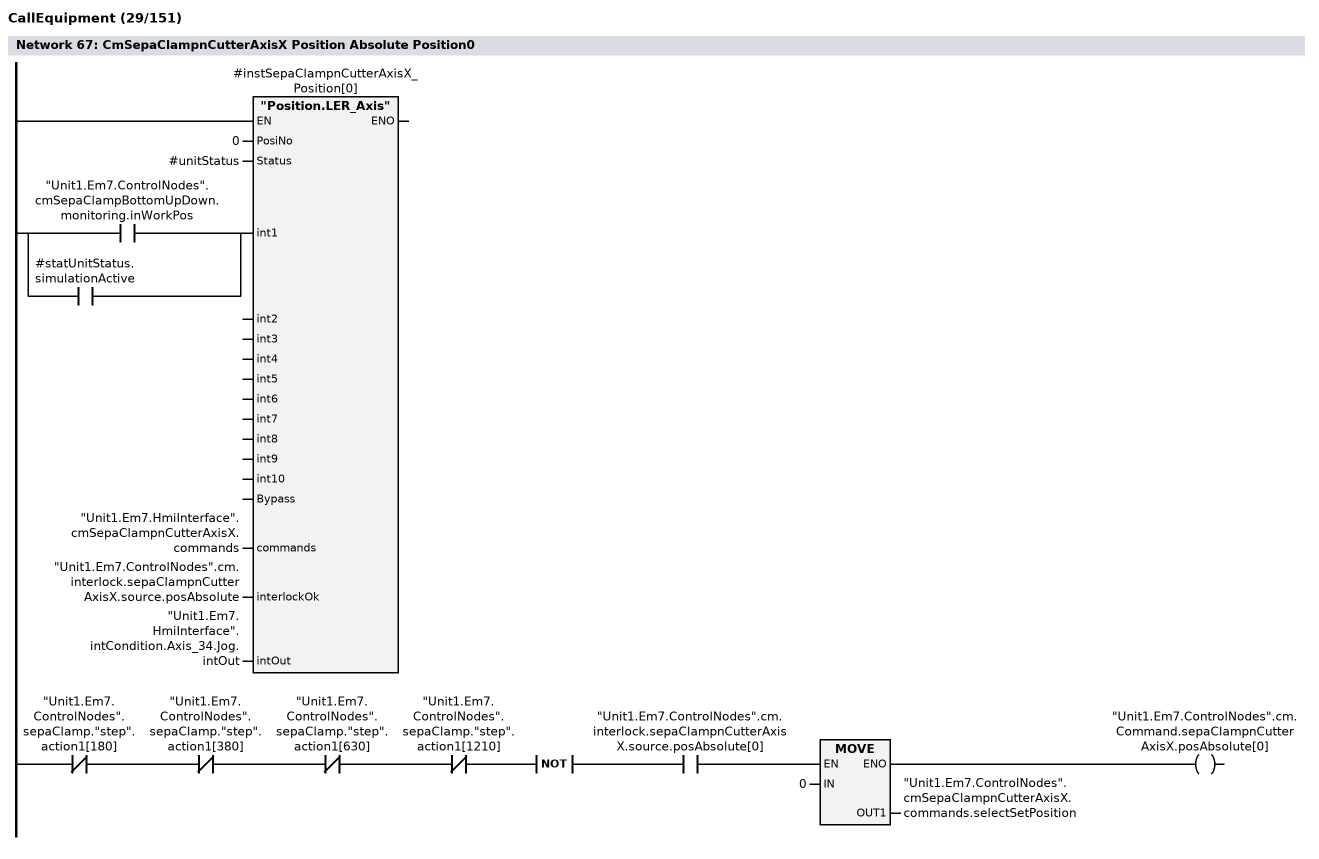
   RUNG wire#powerrail
      #instSepaClampnCutterAxisX_Position[0](int1 := wire#w1, PosiNo := 0, Status := #unitStatus, int2 :=, int3 :=, int4 :=, int5 :=, int6 :=, int7 :=, int8 :=, int9 :=, int10 :=, Bypass :=, commands := "Unit1.Em7.HmiInterface".cmSepaClampnCutterAxisX.commands, interlockOk := "Unit1.Em7.ControlNodes".cm.interlock.sepaClampnCutterAxisX.source.posAbsolute, intOut := "Unit1.Em7.HmiInterface".intCondition.Axis_34.Jog.intOut)
   END_RUNG
   RUNG wire#powerrail
      Contact( "Unit1.Em7.ControlNodes".cmSepaClampBottomUpDown.monitoring.inWorkPos )
   END_RUNG wire#w1
   RUNG wire#powerrail
      Contact( #statUnitStatus.simulationActive )
   END_RUNG wire#w1
   RUNG wire#powerrail
      I_Contact( "Unit1.Em7.ControlNodes".sepaClamp."step".action1[180] )
      I_Contact( "Unit1.Em7.ControlNodes".sepaClamp."step".action1[380] )
      I_Contact( "Unit1.Em7.ControlNodes".sepaClamp."step".action1[630] )
      I_Contact( "Unit1.Em7.ControlNodes".sepaClamp."step".action1[1210] )
      Not()
      Contact( "Unit1.Em7.ControlNodes".cm.interlock.sepaClampnCutterAxisX.source.posAbsolute[0] )
      Move(in := 0, out1 => "Unit1.Em7.ControlNodes".cmSepaClampnCutterAxisX.commands.selectSetPosition)
      Coil( "Unit1.Em7.ControlNodes".cm.Command.sepaClampnCutterAxisX.posAbsolute[0] )
   END_RUNG
   // the same network as SCL:
   #instSepaClampnCutterAxisX_Position[0](PosiNo := 0,   // "Position.LER_Axis"
                           Status := #unitStatus,
                           int1 := "Unit1.Em7.ControlNodes".cmSepaClampBottomUpDown.monitoring.inWorkPos OR #statUnitStatus.simulationActive,
                           commands := "Unit1.Em7.HmiInterface".cmSepaClampnCutterAxisX.commands,
                           interlockOk := "Unit1.Em7.ControlNodes".cm.interlock.sepaClampnCutterAxisX.source.posAbsolute,
                           intOut := "Unit1.Em7.HmiInterface".intCondition.Axis_34.Jog.intOut);
   #_w1 := NOT (NOT "Unit1.Em7.ControlNodes".sepaClamp."step".action1[180] AND NOT "Unit1.Em7.ControlNodes".sepaClamp."step".action1[380] AND NOT "Unit1.Em7.ControlNodes".sepaClamp."step".action1[630] AND NOT "Unit1.Em7.ControlNodes".sepaClamp."step".action1[1210]) AND "Unit1.Em7.ControlNodes".cm.interlock.sepaClampnCutterAxisX.source.posAbsolute[0];
   IF #_w1 THEN "Unit1.Em7.ControlNodes".cmSepaClampnCutterAxisX.commands.selectSetPosition := 0; END_IF;
   "Unit1.Em7.ControlNodes".cm.Command.sepaClampnCutterAxisX.posAbsolute[0] := #_w1;
END_REGION

REGION Network 68: CmSepaClampnCutterAxisX Position Absolute Position1
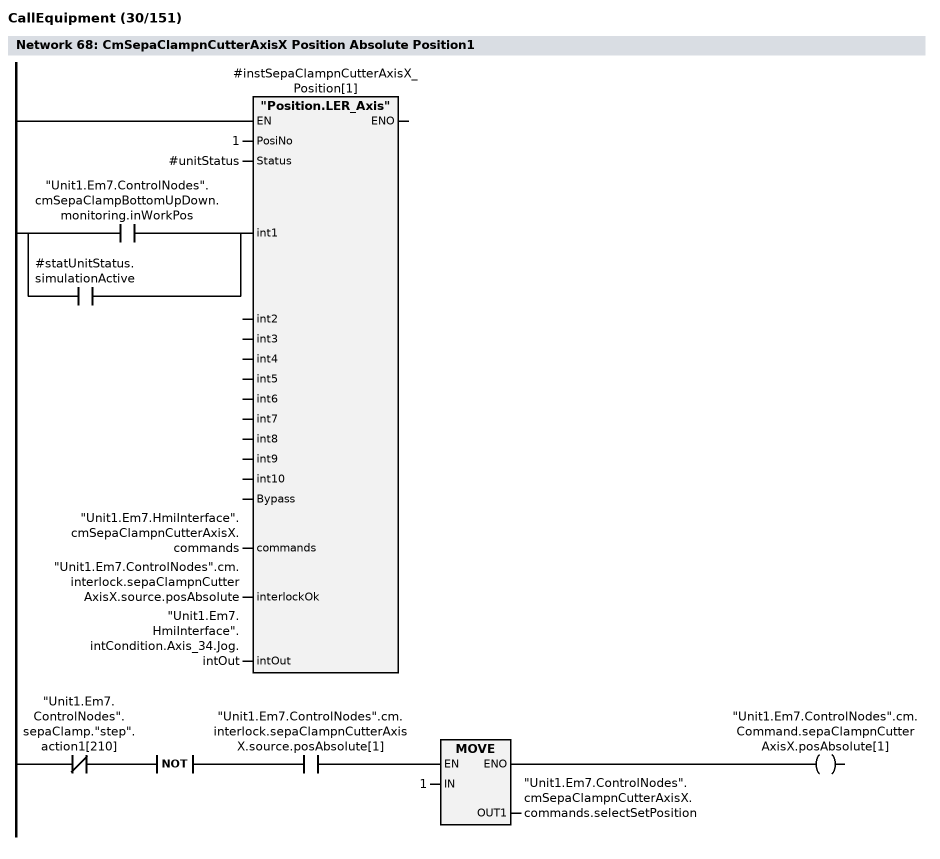
   RUNG wire#powerrail
      #instSepaClampnCutterAxisX_Position[1](int1 := wire#w1, PosiNo := 1, Status := #unitStatus, int2 :=, int3 :=, int4 :=, int5 :=, int6 :=, int7 :=, int8 :=, int9 :=, int10 :=, Bypass :=, commands := "Unit1.Em7.HmiInterface".cmSepaClampnCutterAxisX.commands, interlockOk := "Unit1.Em7.ControlNodes".cm.interlock.sepaClampnCutterAxisX.source.posAbsolute, intOut := "Unit1.Em7.HmiInterface".intCondition.Axis_34.Jog.intOut)
   END_RUNG
   RUNG wire#powerrail
      Contact( "Unit1.Em7.ControlNodes".cmSepaClampBottomUpDown.monitoring.inWorkPos )
   END_RUNG wire#w1
   RUNG wire#powerrail
      Contact( #statUnitStatus.simulationActive )
   END_RUNG wire#w1
   RUNG wire#powerrail
      I_Contact( "Unit1.Em7.ControlNodes".sepaClamp."step".action1[210] )
      Not()
      Contact( "Unit1.Em7.ControlNodes".cm.interlock.sepaClampnCutterAxisX.source.posAbsolute[1] )
      Move(in := 1, out1 => "Unit1.Em7.ControlNodes".cmSepaClampnCutterAxisX.commands.selectSetPosition)
      Coil( "Unit1.Em7.ControlNodes".cm.Command.sepaClampnCutterAxisX.posAbsolute[1] )
   END_RUNG
   // the same network as SCL:
   #instSepaClampnCutterAxisX_Position[1](PosiNo := 1,   // "Position.LER_Axis"
                           Status := #unitStatus,
                           int1 := "Unit1.Em7.ControlNodes".cmSepaClampBottomUpDown.monitoring.inWorkPos OR #statUnitStatus.simulationActive,
                           commands := "Unit1.Em7.HmiInterface".cmSepaClampnCutterAxisX.commands,
                           interlockOk := "Unit1.Em7.ControlNodes".cm.interlock.sepaClampnCutterAxisX.source.posAbsolute,
                           intOut := "Unit1.Em7.HmiInterface".intCondition.Axis_34.Jog.intOut);
   #_w1 := NOT (NOT "Unit1.Em7.ControlNodes".sepaClamp."step".action1[210]) AND "Unit1.Em7.ControlNodes".cm.interlock.sepaClampnCutterAxisX.source.posAbsolute[1];
   IF #_w1 THEN "Unit1.Em7.ControlNodes".cmSepaClampnCutterAxisX.commands.selectSetPosition := 1; END_IF;
   "Unit1.Em7.ControlNodes".cm.Command.sepaClampnCutterAxisX.posAbsolute[1] := #_w1;
END_REGION

REGION Network 69: CmSepaClampnCutterAxisX Position Absolute Position2
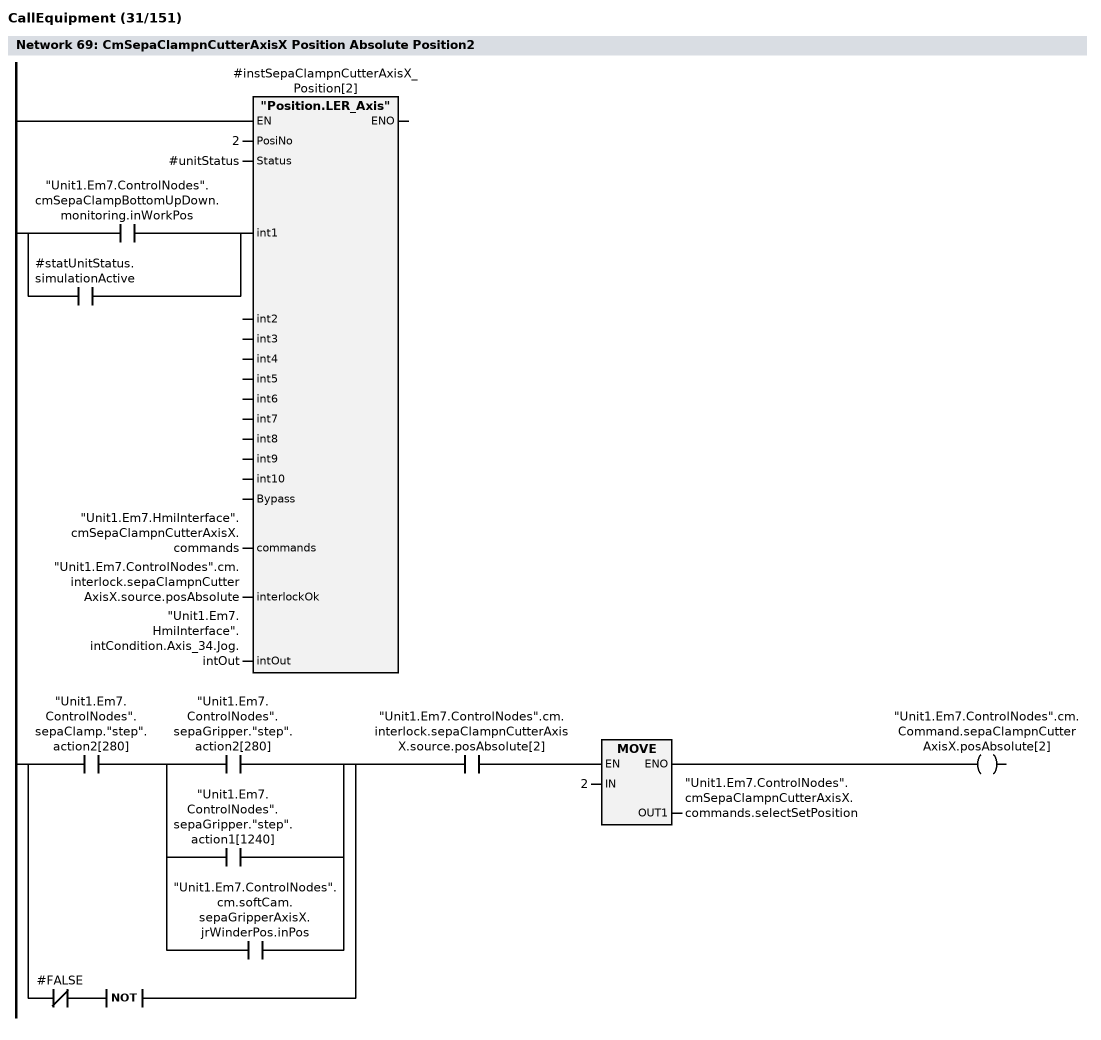
   RUNG wire#powerrail
      #instSepaClampnCutterAxisX_Position[2](int1 := wire#w1, PosiNo := 2, Status := #unitStatus, int2 :=, int3 :=, int4 :=, int5 :=, int6 :=, int7 :=, int8 :=, int9 :=, int10 :=, Bypass :=, commands := "Unit1.Em7.HmiInterface".cmSepaClampnCutterAxisX.commands, interlockOk := "Unit1.Em7.ControlNodes".cm.interlock.sepaClampnCutterAxisX.source.posAbsolute, intOut := "Unit1.Em7.HmiInterface".intCondition.Axis_34.Jog.intOut)
   END_RUNG
   RUNG wire#powerrail
      Contact( "Unit1.Em7.ControlNodes".cmSepaClampBottomUpDown.monitoring.inWorkPos )
   END_RUNG wire#w1
   RUNG wire#powerrail
      Contact( #statUnitStatus.simulationActive )
   END_RUNG wire#w1
   RUNG wire#powerrail
      Contact( "Unit1.Em7.ControlNodes".sepaClamp."step".action2[280] )
      wire#w2
      Contact( "Unit1.Em7.ControlNodes".sepaGripper."step".action2[280] )
      wire#w3
      Contact( "Unit1.Em7.ControlNodes".cm.interlock.sepaClampnCutterAxisX.source.posAbsolute[2] )
      Move(in := 2, out1 => "Unit1.Em7.ControlNodes".cmSepaClampnCutterAxisX.commands.selectSetPosition)
      Coil( "Unit1.Em7.ControlNodes".cm.Command.sepaClampnCutterAxisX.posAbsolute[2] )
   END_RUNG
   RUNG wire#w2
      Contact( "Unit1.Em7.ControlNodes".sepaGripper."step".action1[1240] )
   END_RUNG wire#w3
   RUNG wire#w2
      Contact( "Unit1.Em7.ControlNodes".cm.softCam.sepaGripperAxisX.jrWinderPos.inPos )
   END_RUNG wire#w3
   RUNG wire#powerrail
      I_Contact( #FALSE )
      Not()
   END_RUNG wire#w3
   // the same network as SCL:
   #instSepaClampnCutterAxisX_Position[2](PosiNo := 2,   // "Position.LER_Axis"
                           Status := #unitStatus,
                           int1 := "Unit1.Em7.ControlNodes".cmSepaClampBottomUpDown.monitoring.inWorkPos OR #statUnitStatus.simulationActive,
                           commands := "Unit1.Em7.HmiInterface".cmSepaClampnCutterAxisX.commands,
                           interlockOk := "Unit1.Em7.ControlNodes".cm.interlock.sepaClampnCutterAxisX.source.posAbsolute,
                           intOut := "Unit1.Em7.HmiInterface".intCondition.Axis_34.Jog.intOut);
   #_w1 := (("Unit1.Em7.ControlNodes".sepaClamp."step".action2[280] AND ("Unit1.Em7.ControlNodes".sepaGripper."step".action2[280] OR "Unit1.Em7.ControlNodes".sepaGripper."step".action1[1240] OR "Unit1.Em7.ControlNodes".cm.softCam.sepaGripperAxisX.jrWinderPos.inPos)) OR NOT (NOT #FALSE)) AND "Unit1.Em7.ControlNodes".cm.interlock.sepaClampnCutterAxisX.source.posAbsolute[2];
   IF #_w1 THEN "Unit1.Em7.ControlNodes".cmSepaClampnCutterAxisX.commands.selectSetPosition := 2; END_IF;
   "Unit1.Em7.ControlNodes".cm.Command.sepaClampnCutterAxisX.posAbsolute[2] := #_w1;
END_REGION

REGION Network 70: CmSepaClampnCutterAxisX Position Absolute Position3
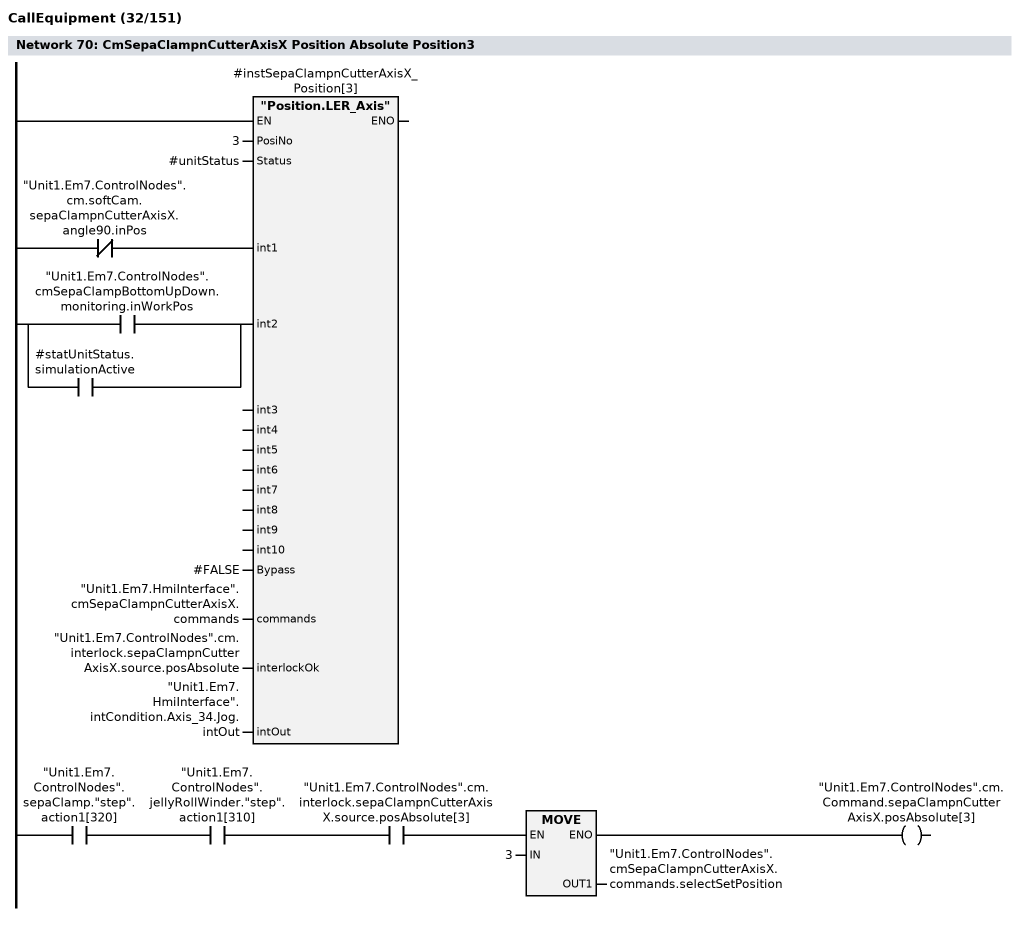
   RUNG wire#powerrail
      #instSepaClampnCutterAxisX_Position[3](int1 := wire#w1, int2 := wire#w2, PosiNo := 3, Status := #unitStatus, int3 :=, int4 :=, int5 :=, int6 :=, int7 :=, int8 :=, int9 :=, int10 :=, Bypass := #FALSE, commands := "Unit1.Em7.HmiInterface".cmSepaClampnCutterAxisX.commands, interlockOk := "Unit1.Em7.ControlNodes".cm.interlock.sepaClampnCutterAxisX.source.posAbsolute, intOut := "Unit1.Em7.HmiInterface".intCondition.Axis_34.Jog.intOut)
   END_RUNG
   RUNG wire#powerrail
      I_Contact( "Unit1.Em7.ControlNodes".cm.softCam.sepaClampnCutterAxisX.angle90.inPos )
   END_RUNG wire#w1
   RUNG wire#powerrail
      Contact( "Unit1.Em7.ControlNodes".cmSepaClampBottomUpDown.monitoring.inWorkPos )
   END_RUNG wire#w2
   RUNG wire#powerrail
      Contact( #statUnitStatus.simulationActive )
   END_RUNG wire#w2
   RUNG wire#powerrail
      Contact( "Unit1.Em7.ControlNodes".sepaClamp."step".action1[320] )
      Contact( "Unit1.Em7.ControlNodes".jellyRollWinder."step".action1[310] )
      Contact( "Unit1.Em7.ControlNodes".cm.interlock.sepaClampnCutterAxisX.source.posAbsolute[3] )
      Move(in := 3, out1 => "Unit1.Em7.ControlNodes".cmSepaClampnCutterAxisX.commands.selectSetPosition)
      Coil( "Unit1.Em7.ControlNodes".cm.Command.sepaClampnCutterAxisX.posAbsolute[3] )
   END_RUNG
   // the same network as SCL:
   #instSepaClampnCutterAxisX_Position[3](PosiNo := 3,   // "Position.LER_Axis"
                           Status := #unitStatus,
                           int1 := NOT "Unit1.Em7.ControlNodes".cm.softCam.sepaClampnCutterAxisX.angle90.inPos,
                           int2 := "Unit1.Em7.ControlNodes".cmSepaClampBottomUpDown.monitoring.inWorkPos OR #statUnitStatus.simulationActive,
                           Bypass := #FALSE,
                           commands := "Unit1.Em7.HmiInterface".cmSepaClampnCutterAxisX.commands,
                           interlockOk := "Unit1.Em7.ControlNodes".cm.interlock.sepaClampnCutterAxisX.source.posAbsolute,
                           intOut := "Unit1.Em7.HmiInterface".intCondition.Axis_34.Jog.intOut);
   #_w1 := "Unit1.Em7.ControlNodes".sepaClamp."step".action1[320] AND "Unit1.Em7.ControlNodes".jellyRollWinder."step".action1[310] AND "Unit1.Em7.ControlNodes".cm.interlock.sepaClampnCutterAxisX.source.posAbsolute[3];
   IF #_w1 THEN "Unit1.Em7.ControlNodes".cmSepaClampnCutterAxisX.commands.selectSetPosition := 3; END_IF;
   "Unit1.Em7.ControlNodes".cm.Command.sepaClampnCutterAxisX.posAbsolute[3] := #_w1;
END_REGION

REGION Network 71: CmSepaClampnCutterAxisX Position Absolute Position4
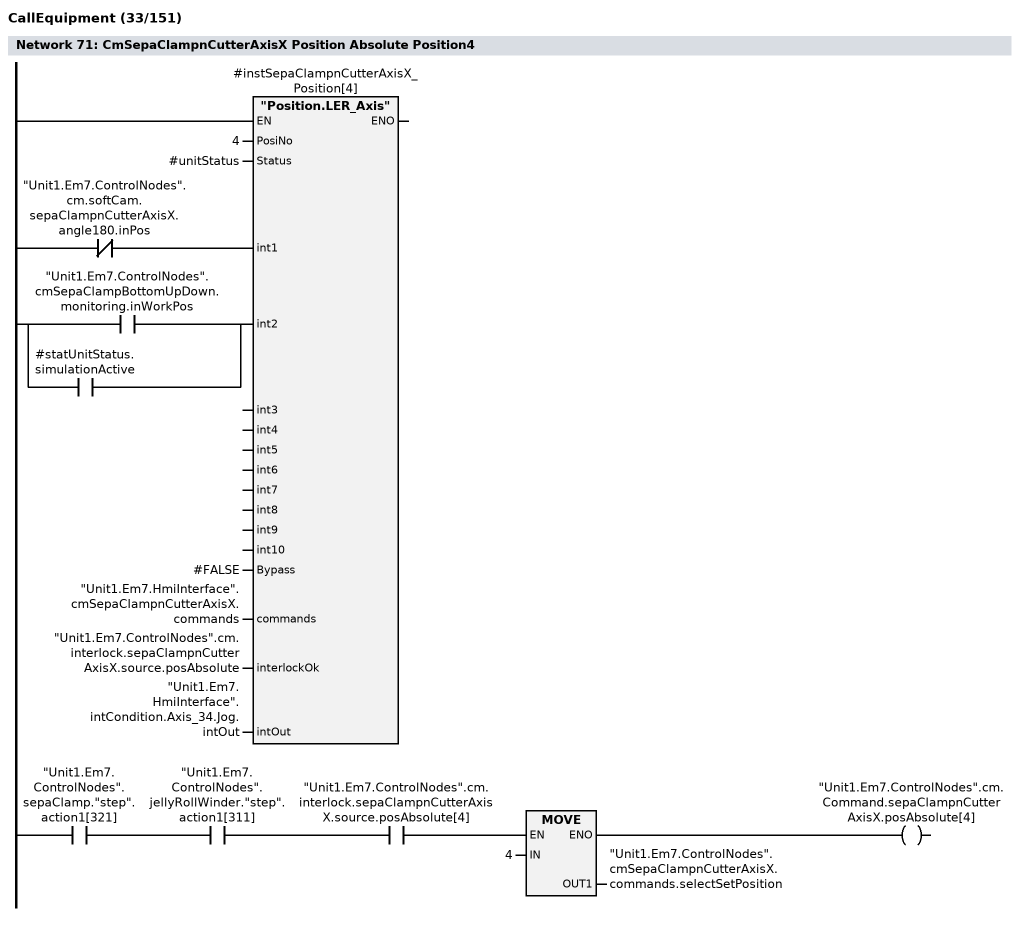
   RUNG wire#powerrail
      #instSepaClampnCutterAxisX_Position[4](int1 := wire#w1, int2 := wire#w2, PosiNo := 4, Status := #unitStatus, int3 :=, int4 :=, int5 :=, int6 :=, int7 :=, int8 :=, int9 :=, int10 :=, Bypass := #FALSE, commands := "Unit1.Em7.HmiInterface".cmSepaClampnCutterAxisX.commands, interlockOk := "Unit1.Em7.ControlNodes".cm.interlock.sepaClampnCutterAxisX.source.posAbsolute, intOut := "Unit1.Em7.HmiInterface".intCondition.Axis_34.Jog.intOut)
   END_RUNG
   RUNG wire#powerrail
      I_Contact( "Unit1.Em7.ControlNodes".cm.softCam.sepaClampnCutterAxisX.angle180.inPos )
   END_RUNG wire#w1
   RUNG wire#powerrail
      Contact( "Unit1.Em7.ControlNodes".cmSepaClampBottomUpDown.monitoring.inWorkPos )
   END_RUNG wire#w2
   RUNG wire#powerrail
      Contact( #statUnitStatus.simulationActive )
   END_RUNG wire#w2
   RUNG wire#powerrail
      Contact( "Unit1.Em7.ControlNodes".sepaClamp."step".action1[321] )
      Contact( "Unit1.Em7.ControlNodes".jellyRollWinder."step".action1[311] )
      Contact( "Unit1.Em7.ControlNodes".cm.interlock.sepaClampnCutterAxisX.source.posAbsolute[4] )
      Move(in := 4, out1 => "Unit1.Em7.ControlNodes".cmSepaClampnCutterAxisX.commands.selectSetPosition)
      Coil( "Unit1.Em7.ControlNodes".cm.Command.sepaClampnCutterAxisX.posAbsolute[4] )
   END_RUNG
   // the same network as SCL:
   #instSepaClampnCutterAxisX_Position[4](PosiNo := 4,   // "Position.LER_Axis"
                           Status := #unitStatus,
                           int1 := NOT "Unit1.Em7.ControlNodes".cm.softCam.sepaClampnCutterAxisX.angle180.inPos,
                           int2 := "Unit1.Em7.ControlNodes".cmSepaClampBottomUpDown.monitoring.inWorkPos OR #statUnitStatus.simulationActive,
                           Bypass := #FALSE,
                           commands := "Unit1.Em7.HmiInterface".cmSepaClampnCutterAxisX.commands,
                           interlockOk := "Unit1.Em7.ControlNodes".cm.interlock.sepaClampnCutterAxisX.source.posAbsolute,
                           intOut := "Unit1.Em7.HmiInterface".intCondition.Axis_34.Jog.intOut);
   #_w1 := "Unit1.Em7.ControlNodes".sepaClamp."step".action1[321] AND "Unit1.Em7.ControlNodes".jellyRollWinder."step".action1[311] AND "Unit1.Em7.ControlNodes".cm.interlock.sepaClampnCutterAxisX.source.posAbsolute[4];
   IF #_w1 THEN "Unit1.Em7.ControlNodes".cmSepaClampnCutterAxisX.commands.selectSetPosition := 4; END_IF;
   "Unit1.Em7.ControlNodes".cm.Command.sepaClampnCutterAxisX.posAbsolute[4] := #_w1;
END_REGION

REGION Network 72: CmSepaClampnCutterAxisX Position Absolute Position5
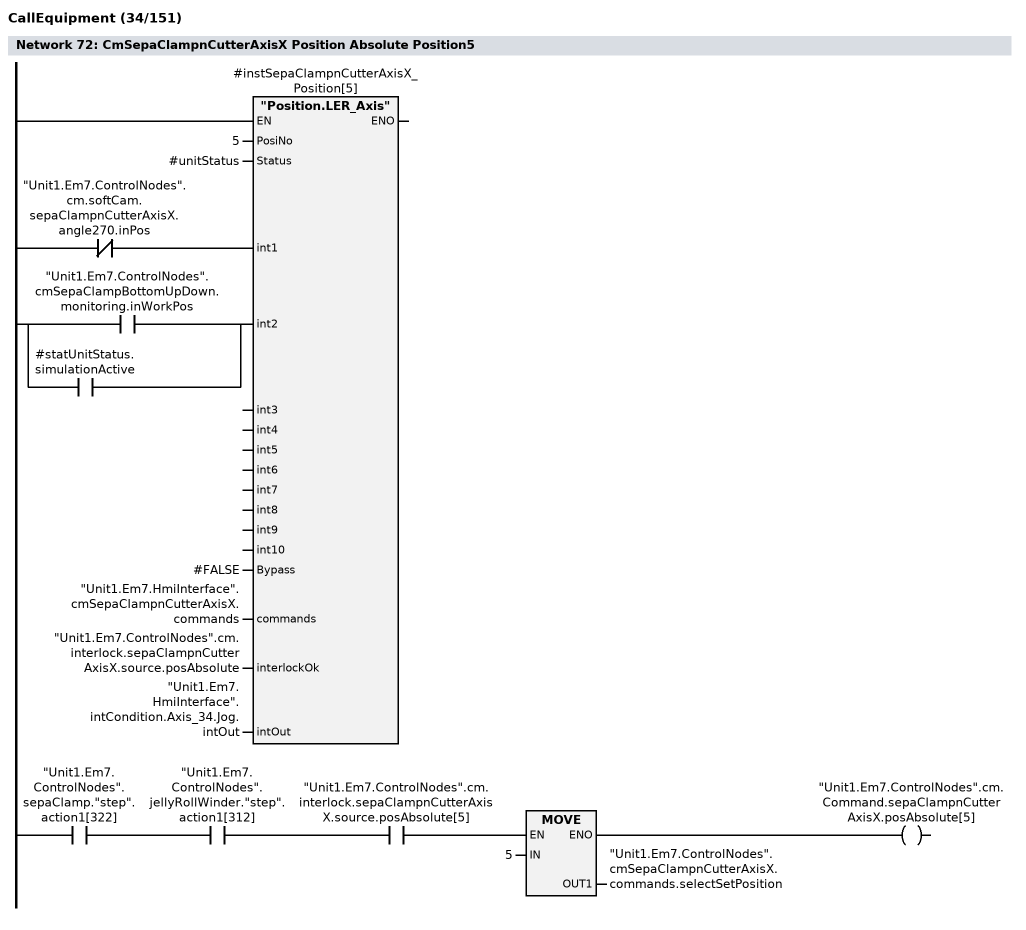
   RUNG wire#powerrail
      #instSepaClampnCutterAxisX_Position[5](int1 := wire#w1, int2 := wire#w2, PosiNo := 5, Status := #unitStatus, int3 :=, int4 :=, int5 :=, int6 :=, int7 :=, int8 :=, int9 :=, int10 :=, Bypass := #FALSE, commands := "Unit1.Em7.HmiInterface".cmSepaClampnCutterAxisX.commands, interlockOk := "Unit1.Em7.ControlNodes".cm.interlock.sepaClampnCutterAxisX.source.posAbsolute, intOut := "Unit1.Em7.HmiInterface".intCondition.Axis_34.Jog.intOut)
   END_RUNG
   RUNG wire#powerrail
      I_Contact( "Unit1.Em7.ControlNodes".cm.softCam.sepaClampnCutterAxisX.angle270.inPos )
   END_RUNG wire#w1
   RUNG wire#powerrail
      Contact( "Unit1.Em7.ControlNodes".cmSepaClampBottomUpDown.monitoring.inWorkPos )
   END_RUNG wire#w2
   RUNG wire#powerrail
      Contact( #statUnitStatus.simulationActive )
   END_RUNG wire#w2
   RUNG wire#powerrail
      Contact( "Unit1.Em7.ControlNodes".sepaClamp."step".action1[322] )
      Contact( "Unit1.Em7.ControlNodes".jellyRollWinder."step".action1[312] )
      Contact( "Unit1.Em7.ControlNodes".cm.interlock.sepaClampnCutterAxisX.source.posAbsolute[5] )
      Move(in := 5, out1 => "Unit1.Em7.ControlNodes".cmSepaClampnCutterAxisX.commands.selectSetPosition)
      Coil( "Unit1.Em7.ControlNodes".cm.Command.sepaClampnCutterAxisX.posAbsolute[5] )
   END_RUNG
   // the same network as SCL:
   #instSepaClampnCutterAxisX_Position[5](PosiNo := 5,   // "Position.LER_Axis"
                           Status := #unitStatus,
                           int1 := NOT "Unit1.Em7.ControlNodes".cm.softCam.sepaClampnCutterAxisX.angle270.inPos,
                           int2 := "Unit1.Em7.ControlNodes".cmSepaClampBottomUpDown.monitoring.inWorkPos OR #statUnitStatus.simulationActive,
                           Bypass := #FALSE,
                           commands := "Unit1.Em7.HmiInterface".cmSepaClampnCutterAxisX.commands,
                           interlockOk := "Unit1.Em7.ControlNodes".cm.interlock.sepaClampnCutterAxisX.source.posAbsolute,
                           intOut := "Unit1.Em7.HmiInterface".intCondition.Axis_34.Jog.intOut);
   #_w1 := "Unit1.Em7.ControlNodes".sepaClamp."step".action1[322] AND "Unit1.Em7.ControlNodes".jellyRollWinder."step".action1[312] AND "Unit1.Em7.ControlNodes".cm.interlock.sepaClampnCutterAxisX.source.posAbsolute[5];
   IF #_w1 THEN "Unit1.Em7.ControlNodes".cmSepaClampnCutterAxisX.commands.selectSetPosition := 5; END_IF;
   "Unit1.Em7.ControlNodes".cm.Command.sepaClampnCutterAxisX.posAbsolute[5] := #_w1;
END_REGION

REGION Network 73: CmSepaClampnCutterAxisX Position Absolute Position6
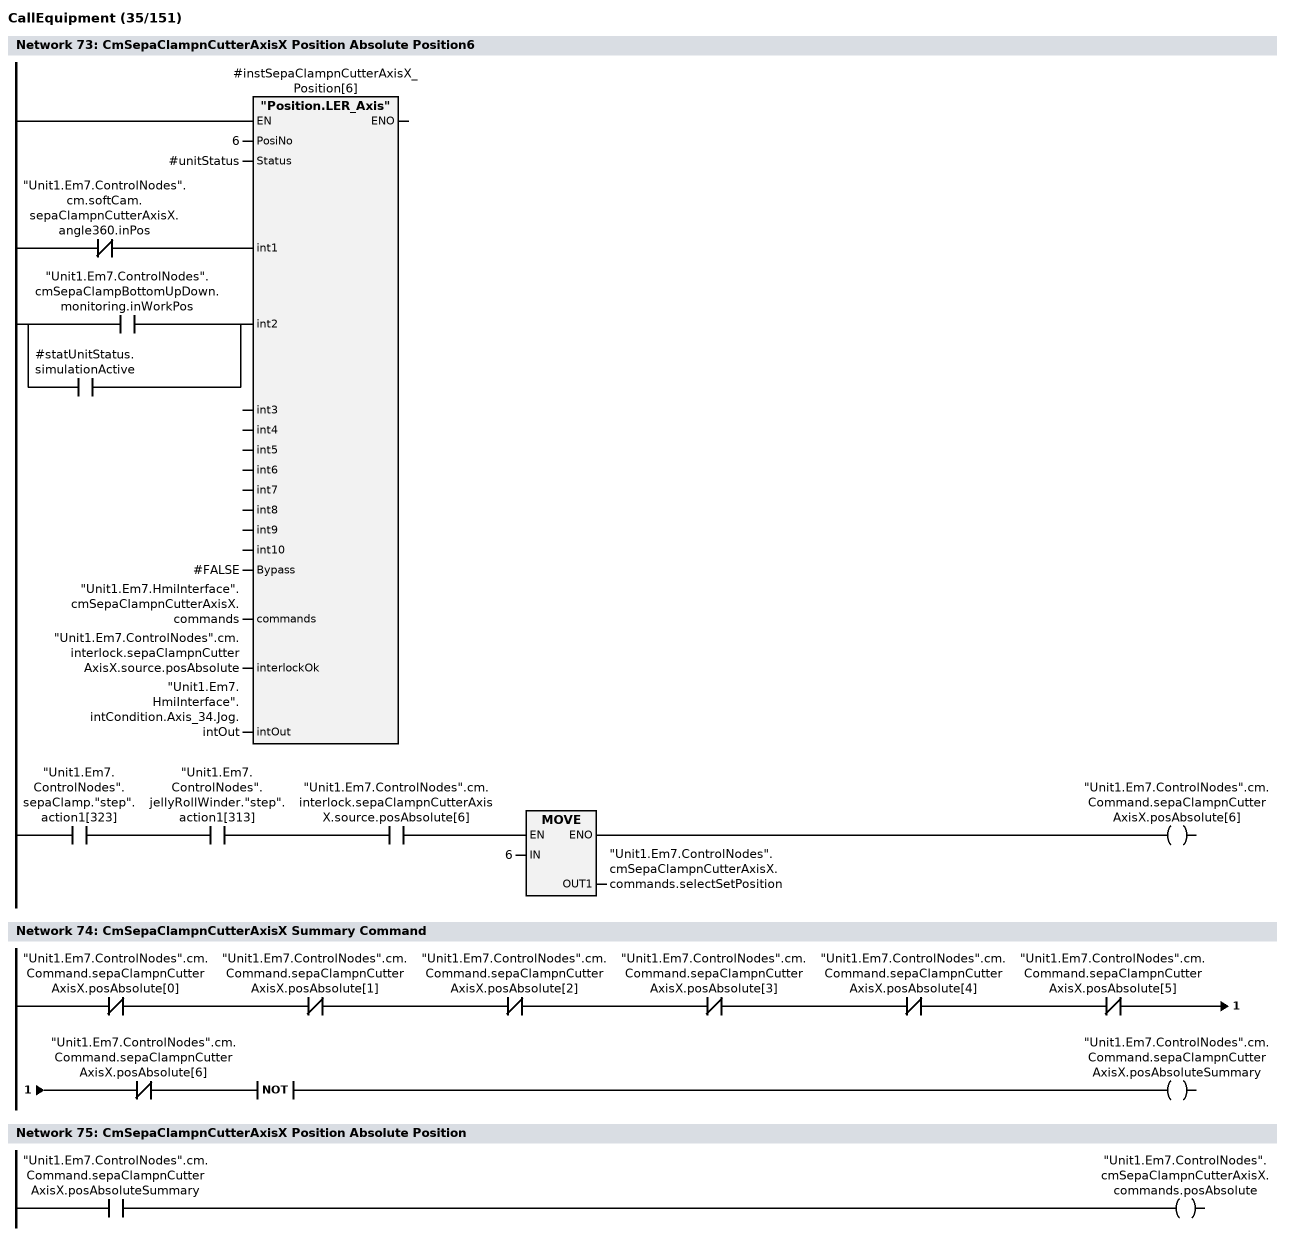
   RUNG wire#powerrail
      #instSepaClampnCutterAxisX_Position[6](int1 := wire#w1, int2 := wire#w2, PosiNo := 6, Status := #unitStatus, int3 :=, int4 :=, int5 :=, int6 :=, int7 :=, int8 :=, int9 :=, int10 :=, Bypass := #FALSE, commands := "Unit1.Em7.HmiInterface".cmSepaClampnCutterAxisX.commands, interlockOk := "Unit1.Em7.ControlNodes".cm.interlock.sepaClampnCutterAxisX.source.posAbsolute, intOut := "Unit1.Em7.HmiInterface".intCondition.Axis_34.Jog.intOut)
   END_RUNG
   RUNG wire#powerrail
      I_Contact( "Unit1.Em7.ControlNodes".cm.softCam.sepaClampnCutterAxisX.angle360.inPos )
   END_RUNG wire#w1
   RUNG wire#powerrail
      Contact( "Unit1.Em7.ControlNodes".cmSepaClampBottomUpDown.monitoring.inWorkPos )
   END_RUNG wire#w2
   RUNG wire#powerrail
      Contact( #statUnitStatus.simulationActive )
   END_RUNG wire#w2
   RUNG wire#powerrail
      Contact( "Unit1.Em7.ControlNodes".sepaClamp."step".action1[323] )
      Contact( "Unit1.Em7.ControlNodes".jellyRollWinder."step".action1[313] )
      Contact( "Unit1.Em7.ControlNodes".cm.interlock.sepaClampnCutterAxisX.source.posAbsolute[6] )
      Move(in := 6, out1 => "Unit1.Em7.ControlNodes".cmSepaClampnCutterAxisX.commands.selectSetPosition)
      Coil( "Unit1.Em7.ControlNodes".cm.Command.sepaClampnCutterAxisX.posAbsolute[6] )
   END_RUNG
   // the same network as SCL:
   #instSepaClampnCutterAxisX_Position[6](PosiNo := 6,   // "Position.LER_Axis"
                           Status := #unitStatus,
                           int1 := NOT "Unit1.Em7.ControlNodes".cm.softCam.sepaClampnCutterAxisX.angle360.inPos,
                           int2 := "Unit1.Em7.ControlNodes".cmSepaClampBottomUpDown.monitoring.inWorkPos OR #statUnitStatus.simulationActive,
                           Bypass := #FALSE,
                           commands := "Unit1.Em7.HmiInterface".cmSepaClampnCutterAxisX.commands,
                           interlockOk := "Unit1.Em7.ControlNodes".cm.interlock.sepaClampnCutterAxisX.source.posAbsolute,
                           intOut := "Unit1.Em7.HmiInterface".intCondition.Axis_34.Jog.intOut);
   #_w1 := "Unit1.Em7.ControlNodes".sepaClamp."step".action1[323] AND "Unit1.Em7.ControlNodes".jellyRollWinder."step".action1[313] AND "Unit1.Em7.ControlNodes".cm.interlock.sepaClampnCutterAxisX.source.posAbsolute[6];
   IF #_w1 THEN "Unit1.Em7.ControlNodes".cmSepaClampnCutterAxisX.commands.selectSetPosition := 6; END_IF;
   "Unit1.Em7.ControlNodes".cm.Command.sepaClampnCutterAxisX.posAbsolute[6] := #_w1;
END_REGION

REGION Network 74: CmSepaClampnCutterAxisX Summary Command
   RUNG wire#powerrail
      I_Contact( "Unit1.Em7.ControlNodes".cm.Command.sepaClampnCutterAxisX.posAbsolute[0] )
      I_Contact( "Unit1.Em7.ControlNodes".cm.Command.sepaClampnCutterAxisX.posAbsolute[1] )
      I_Contact( "Unit1.Em7.ControlNodes".cm.Command.sepaClampnCutterAxisX.posAbsolute[2] )
      I_Contact( "Unit1.Em7.ControlNodes".cm.Command.sepaClampnCutterAxisX.posAbsolute[3] )
      I_Contact( "Unit1.Em7.ControlNodes".cm.Command.sepaClampnCutterAxisX.posAbsolute[4] )
      I_Contact( "Unit1.Em7.ControlNodes".cm.Command.sepaClampnCutterAxisX.posAbsolute[5] )
      I_Contact( "Unit1.Em7.ControlNodes".cm.Command.sepaClampnCutterAxisX.posAbsolute[6] )
      Not()
      Coil( "Unit1.Em7.ControlNodes".cm.Command.sepaClampnCutterAxisX.posAbsoluteSummary )
   END_RUNG
   // the same network as SCL:
   "Unit1.Em7.ControlNodes".cm.Command.sepaClampnCutterAxisX.posAbsoluteSummary := NOT (NOT "Unit1.Em7.ControlNodes".cm.Command.sepaClampnCutterAxisX.posAbsolute[0] AND NOT "Unit1.Em7.ControlNodes".cm.Command.sepaClampnCutterAxisX.posAbsolute[1] AND NOT "Unit1.Em7.ControlNodes".cm.Command.sepaClampnCutterAxisX.posAbsolute[2] AND NOT "Unit1.Em7.ControlNodes".cm.Command.sepaClampnCutterAxisX.posAbsolute[3] AND NOT "Unit1.Em7.ControlNodes".cm.Command.sepaClampnCutterAxisX.posAbsolute[4] AND NOT "Unit1.Em7.ControlNodes".cm.Command.sepaClampnCutterAxisX.posAbsolute[5] AND NOT "Unit1.Em7.ControlNodes".cm.Command.sepaClampnCutterAxisX.posAbsolute[6]);
END_REGION

REGION Network 75: CmSepaClampnCutterAxisX Position Absolute Position
   RUNG wire#powerrail
      Contact( "Unit1.Em7.ControlNodes".cm.Command.sepaClampnCutterAxisX.posAbsoluteSummary )
      Coil( "Unit1.Em7.ControlNodes".cmSepaClampnCutterAxisX.commands.posAbsolute )
   END_RUNG
   // the same network as SCL:
   "Unit1.Em7.ControlNodes".cmSepaClampnCutterAxisX.commands.posAbsolute := "Unit1.Em7.ControlNodes".cm.Command.sepaClampnCutterAxisX.posAbsoluteSummary;
END_REGION

REGION Network 76: CmSepaClampnCutterAxisX Interlock Summary
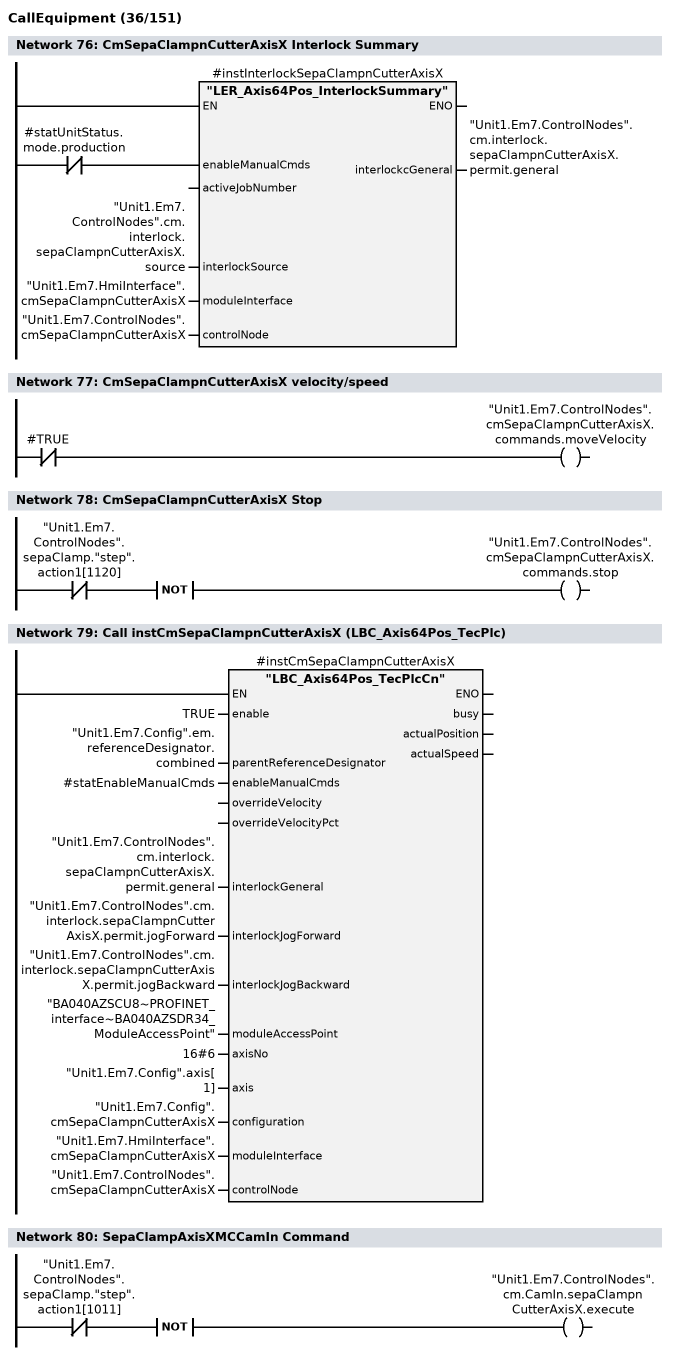
   RUNG wire#powerrail
      #instInterlockSepaClampnCutterAxisX(enableManualCmds := wire#w1, activeJobNumber :=, interlockSource := "Unit1.Em7.ControlNodes".cm.interlock.sepaClampnCutterAxisX.source, moduleInterface := "Unit1.Em7.HmiInterface".cmSepaClampnCutterAxisX, controlNode := "Unit1.Em7.ControlNodes".cmSepaClampnCutterAxisX, interlockcGeneral => "Unit1.Em7.ControlNodes".cm.interlock.sepaClampnCutterAxisX.permit.general)
   END_RUNG
   RUNG wire#powerrail
      I_Contact( #statUnitStatus.mode.production )
   END_RUNG wire#w1
   // the same network as SCL:
   #instInterlockSepaClampnCutterAxisX(enableManualCmds := NOT #statUnitStatus.mode.production,   // "LER_Axis64Pos_InterlockSummary"
                           interlockSource := "Unit1.Em7.ControlNodes".cm.interlock.sepaClampnCutterAxisX.source,
                           moduleInterface := "Unit1.Em7.HmiInterface".cmSepaClampnCutterAxisX,
                           controlNode := "Unit1.Em7.ControlNodes".cmSepaClampnCutterAxisX,
                           interlockcGeneral => "Unit1.Em7.ControlNodes".cm.interlock.sepaClampnCutterAxisX.permit.general);
END_REGION

REGION Network 77: CmSepaClampnCutterAxisX velocity/speed
   RUNG wire#powerrail
      I_Contact( #TRUE )
      Coil( "Unit1.Em7.ControlNodes".cmSepaClampnCutterAxisX.commands.moveVelocity )
   END_RUNG
   // the same network as SCL:
   "Unit1.Em7.ControlNodes".cmSepaClampnCutterAxisX.commands.moveVelocity := NOT #TRUE;
END_REGION

REGION Network 78: CmSepaClampnCutterAxisX Stop
   RUNG wire#powerrail
      I_Contact( "Unit1.Em7.ControlNodes".sepaClamp."step".action1[1120] )
      Not()
      Coil( "Unit1.Em7.ControlNodes".cmSepaClampnCutterAxisX.commands.stop )
   END_RUNG
   // the same network as SCL:
   "Unit1.Em7.ControlNodes".cmSepaClampnCutterAxisX.commands.stop := NOT (NOT "Unit1.Em7.ControlNodes".sepaClamp."step".action1[1120]);
END_REGION

REGION Network 79: Call instCmSepaClampnCutterAxisX (LBC_Axis64Pos_TecPlc)
   RUNG wire#powerrail
      #instCmSepaClampnCutterAxisX(enable := TRUE, parentReferenceDesignator := "Unit1.Em7.Config".em.referenceDesignator.combined, enableManualCmds := #statEnableManualCmds, overrideVelocity :=, overrideVelocityPct :=, interlockGeneral := "Unit1.Em7.ControlNodes".cm.interlock.sepaClampnCutterAxisX.permit.general, interlockJogForward := "Unit1.Em7.ControlNodes".cm.interlock.sepaClampnCutterAxisX.permit.jogForward, interlockJogBackward := "Unit1.Em7.ControlNodes".cm.interlock.sepaClampnCutterAxisX.permit.jogBackward, moduleAccessPoint := "BA040AZSCU8~PROFINET_interface~BA040AZSDR34_ModuleAccessPoint", axisNo := 16#6, axis := "Unit1.Em7.Config".axis[1], configuration := "Unit1.Em7.Config".cmSepaClampnCutterAxisX, moduleInterface := "Unit1.Em7.HmiInterface".cmSepaClampnCutterAxisX, controlNode := "Unit1.Em7.ControlNodes".cmSepaClampnCutterAxisX, busy =>, actualPosition =>, actualSpeed =>)
   END_RUNG
   // the same network as SCL:
   #instCmSepaClampnCutterAxisX(enable := TRUE,   // "LBC_Axis64Pos_TecPlcCn"
                           parentReferenceDesignator := "Unit1.Em7.Config".em.referenceDesignator.combined,
                           enableManualCmds := #statEnableManualCmds,
                           interlockGeneral := "Unit1.Em7.ControlNodes".cm.interlock.sepaClampnCutterAxisX.permit.general,
                           interlockJogForward := "Unit1.Em7.ControlNodes".cm.interlock.sepaClampnCutterAxisX.permit.jogForward,
                           interlockJogBackward := "Unit1.Em7.ControlNodes".cm.interlock.sepaClampnCutterAxisX.permit.jogBackward,
                           moduleAccessPoint := "BA040AZSCU8~PROFINET_interface~BA040AZSDR34_ModuleAccessPoint",
                           axisNo := 16#6,
                           axis := "Unit1.Em7.Config".axis[1],
                           configuration := "Unit1.Em7.Config".cmSepaClampnCutterAxisX,
                           moduleInterface := "Unit1.Em7.HmiInterface".cmSepaClampnCutterAxisX,
                           controlNode := "Unit1.Em7.ControlNodes".cmSepaClampnCutterAxisX);
END_REGION

REGION Network 80: SepaClampAxisXMCCamIn Command
   RUNG wire#powerrail
      I_Contact( "Unit1.Em7.ControlNodes".sepaClamp."step".action1[1011] )
      Not()
      Coil( "Unit1.Em7.ControlNodes".cm.CamIn.sepaClampnCutterAxisX.execute )
   END_RUNG
   // the same network as SCL:
   "Unit1.Em7.ControlNodes".cm.CamIn.sepaClampnCutterAxisX.execute := NOT (NOT "Unit1.Em7.ControlNodes".sepaClamp."step".action1[1011]);
END_REGION

REGION Network 81: Call instSepaClampAxisXMCCamIn
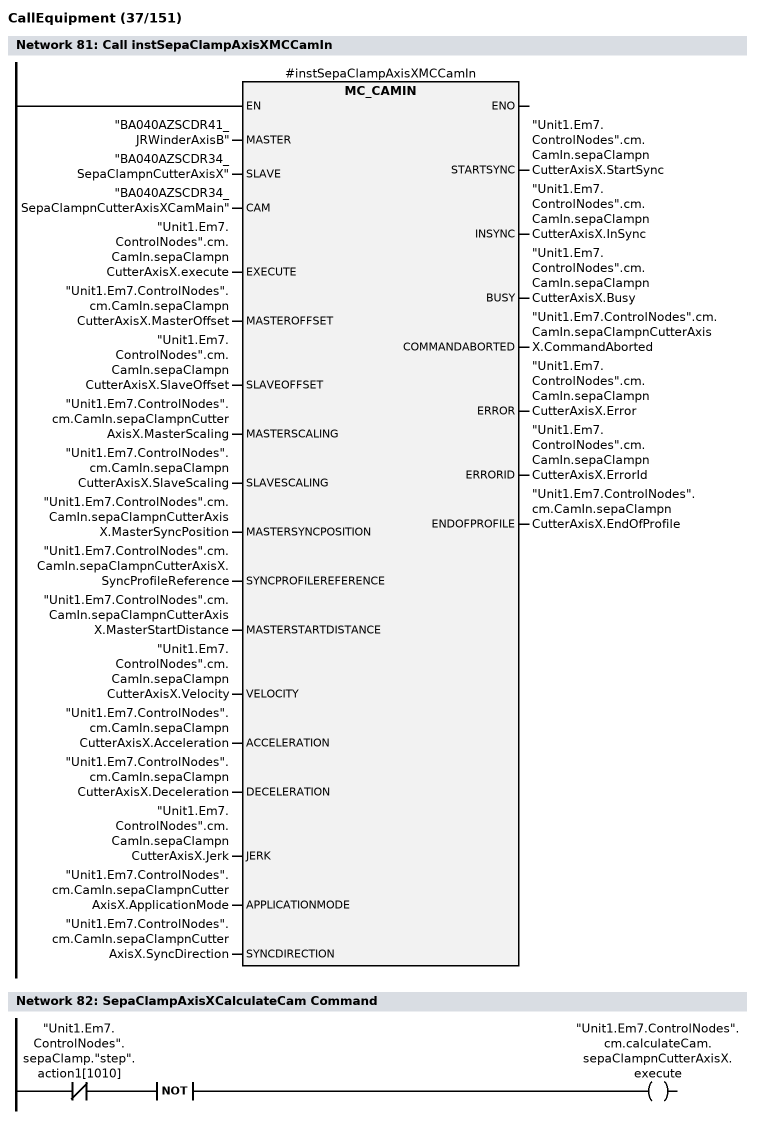
   RUNG wire#powerrail
      #instSepaClampAxisXMCCamIn.MC_CAMIN(Master := "BA040AZSCDR41_JRWinderAxisB", Slave := "BA040AZSCDR34_SepaClampnCutterAxisX", Cam := "BA040AZSCDR34_SepaClampnCutterAxisXCamMain", Execute := "Unit1.Em7.ControlNodes".cm.CamIn.sepaClampnCutterAxisX.execute, MasterOffset := "Unit1.Em7.ControlNodes".cm.CamIn.sepaClampnCutterAxisX.MasterOffset, SlaveOffset := "Unit1.Em7.ControlNodes".cm.CamIn.sepaClampnCutterAxisX.SlaveOffset, MasterScaling := "Unit1.Em7.ControlNodes".cm.CamIn.sepaClampnCutterAxisX.MasterScaling, SlaveScaling := "Unit1.Em7.ControlNodes".cm.CamIn.sepaClampnCutterAxisX.SlaveScaling, MasterSyncPosition := "Unit1.Em7.ControlNodes".cm.CamIn.sepaClampnCutterAxisX.MasterSyncPosition, SyncProfileReference := "Unit1.Em7.ControlNodes".cm.CamIn.sepaClampnCutterAxisX.SyncProfileReference, MasterStartDistance := "Unit1.Em7.ControlNodes".cm.CamIn.sepaClampnCutterAxisX.MasterStartDistance, Velocity := "Unit1.Em7.ControlNodes".cm.CamIn.sepaClampnCutterAxisX.Velocity, Acceleration := "Unit1.Em7.ControlNodes".cm.CamIn.sepaClampnCutterAxisX.Acceleration, Deceleration := "Unit1.Em7.ControlNodes".cm.CamIn.sepaClampnCutterAxisX.Deceleration, Jerk := "Unit1.Em7.ControlNodes".cm.CamIn.sepaClampnCutterAxisX.Jerk, ApplicationMode := "Unit1.Em7.ControlNodes".cm.CamIn.sepaClampnCutterAxisX.ApplicationMode, SyncDirection := "Unit1.Em7.ControlNodes".cm.CamIn.sepaClampnCutterAxisX.SyncDirection, StartSync => "Unit1.Em7.ControlNodes".cm.CamIn.sepaClampnCutterAxisX.StartSync, InSync => "Unit1.Em7.ControlNodes".cm.CamIn.sepaClampnCutterAxisX.InSync, Busy => "Unit1.Em7.ControlNodes".cm.CamIn.sepaClampnCutterAxisX.Busy, CommandAborted => "Unit1.Em7.ControlNodes".cm.CamIn.sepaClampnCutterAxisX.CommandAborted, Error => "Unit1.Em7.ControlNodes".cm.CamIn.sepaClampnCutterAxisX.Error, ErrorId => "Unit1.Em7.ControlNodes".cm.CamIn.sepaClampnCutterAxisX.ErrorId, EndOfProfile => "Unit1.Em7.ControlNodes".cm.CamIn.sepaClampnCutterAxisX.EndOfProfile)
   END_RUNG
   // the same network as SCL:
   #instSepaClampAxisXMCCamIn(Master := "BA040AZSCDR41_JRWinderAxisB",   // MC_CAMIN
                           Slave := "BA040AZSCDR34_SepaClampnCutterAxisX",
                           Cam := "BA040AZSCDR34_SepaClampnCutterAxisXCamMain",
                           Execute := "Unit1.Em7.ControlNodes".cm.CamIn.sepaClampnCutterAxisX.execute,
                           MasterOffset := "Unit1.Em7.ControlNodes".cm.CamIn.sepaClampnCutterAxisX.MasterOffset,
                           SlaveOffset := "Unit1.Em7.ControlNodes".cm.CamIn.sepaClampnCutterAxisX.SlaveOffset,
                           MasterScaling := "Unit1.Em7.ControlNodes".cm.CamIn.sepaClampnCutterAxisX.MasterScaling,
                           SlaveScaling := "Unit1.Em7.ControlNodes".cm.CamIn.sepaClampnCutterAxisX.SlaveScaling,
                           MasterSyncPosition := "Unit1.Em7.ControlNodes".cm.CamIn.sepaClampnCutterAxisX.MasterSyncPosition,
                           SyncProfileReference := "Unit1.Em7.ControlNodes".cm.CamIn.sepaClampnCutterAxisX.SyncProfileReference,
                           MasterStartDistance := "Unit1.Em7.ControlNodes".cm.CamIn.sepaClampnCutterAxisX.MasterStartDistance,
                           Velocity := "Unit1.Em7.ControlNodes".cm.CamIn.sepaClampnCutterAxisX.Velocity,
                           Acceleration := "Unit1.Em7.ControlNodes".cm.CamIn.sepaClampnCutterAxisX.Acceleration,
                           Deceleration := "Unit1.Em7.ControlNodes".cm.CamIn.sepaClampnCutterAxisX.Deceleration,
                           Jerk := "Unit1.Em7.ControlNodes".cm.CamIn.sepaClampnCutterAxisX.Jerk,
                           ApplicationMode := "Unit1.Em7.ControlNodes".cm.CamIn.sepaClampnCutterAxisX.ApplicationMode,
                           SyncDirection := "Unit1.Em7.ControlNodes".cm.CamIn.sepaClampnCutterAxisX.SyncDirection,
                           StartSync => "Unit1.Em7.ControlNodes".cm.CamIn.sepaClampnCutterAxisX.StartSync,
                           InSync => "Unit1.Em7.ControlNodes".cm.CamIn.sepaClampnCutterAxisX.InSync,
                           Busy => "Unit1.Em7.ControlNodes".cm.CamIn.sepaClampnCutterAxisX.Busy,
                           CommandAborted => "Unit1.Em7.ControlNodes".cm.CamIn.sepaClampnCutterAxisX.CommandAborted,
                           Error => "Unit1.Em7.ControlNodes".cm.CamIn.sepaClampnCutterAxisX.Error,
                           ErrorId => "Unit1.Em7.ControlNodes".cm.CamIn.sepaClampnCutterAxisX.ErrorId,
                           EndOfProfile => "Unit1.Em7.ControlNodes".cm.CamIn.sepaClampnCutterAxisX.EndOfProfile);
END_REGION

REGION Network 82: SepaClampAxisXCalculateCam Command
   RUNG wire#powerrail
      I_Contact( "Unit1.Em7.ControlNodes".sepaClamp."step".action1[1010] )
      Not()
      Coil( "Unit1.Em7.ControlNodes".cm.calculateCam.sepaClampnCutterAxisX.execute )
   END_RUNG
   // the same network as SCL:
   "Unit1.Em7.ControlNodes".cm.calculateCam.sepaClampnCutterAxisX.execute := NOT (NOT "Unit1.Em7.ControlNodes".sepaClamp."step".action1[1010]);
END_REGION

REGION Network 83: Call instSepaClampAxisXCalculateCam
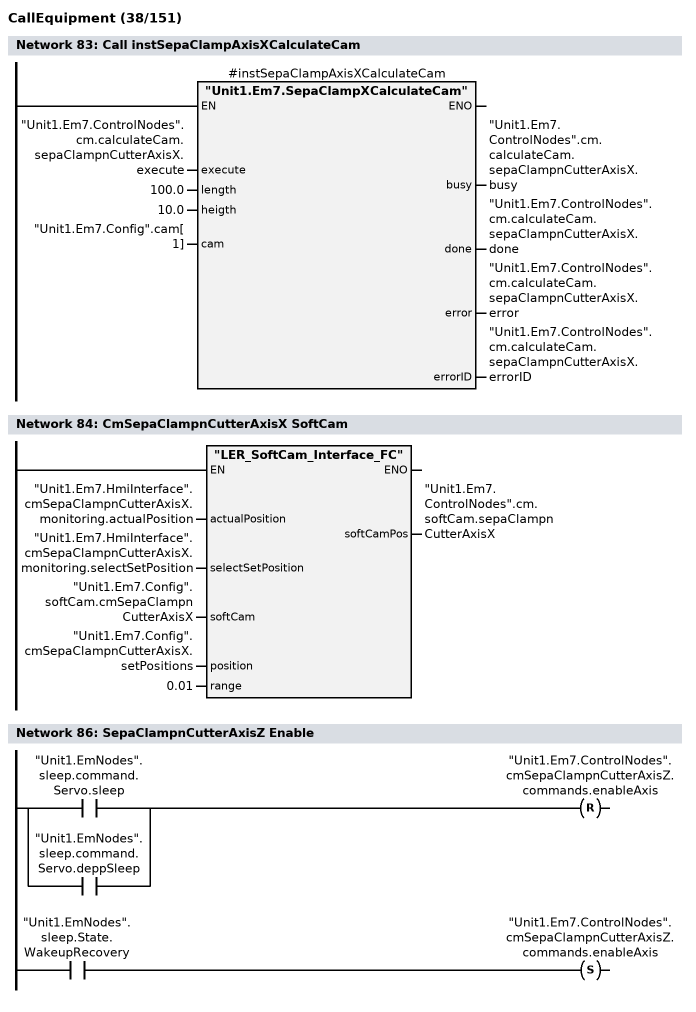
   RUNG wire#powerrail
      #instSepaClampAxisXCalculateCam(execute := "Unit1.Em7.ControlNodes".cm.calculateCam.sepaClampnCutterAxisX.execute, length := 100.0, heigth := 10.0, cam := "Unit1.Em7.Config".cam[1], busy => "Unit1.Em7.ControlNodes".cm.calculateCam.sepaClampnCutterAxisX.busy, done => "Unit1.Em7.ControlNodes".cm.calculateCam.sepaClampnCutterAxisX.done, error => "Unit1.Em7.ControlNodes".cm.calculateCam.sepaClampnCutterAxisX.error, errorID => "Unit1.Em7.ControlNodes".cm.calculateCam.sepaClampnCutterAxisX.errorID)
   END_RUNG
   // the same network as SCL:
   #instSepaClampAxisXCalculateCam(execute := "Unit1.Em7.ControlNodes".cm.calculateCam.sepaClampnCutterAxisX.execute,   // "Unit1.Em7.SepaClampXCalculateCam"
                           length := 100.0,
                           heigth := 10.0,
                           cam := "Unit1.Em7.Config".cam[1],
                           busy => "Unit1.Em7.ControlNodes".cm.calculateCam.sepaClampnCutterAxisX.busy,
                           done => "Unit1.Em7.ControlNodes".cm.calculateCam.sepaClampnCutterAxisX.done,
                           error => "Unit1.Em7.ControlNodes".cm.calculateCam.sepaClampnCutterAxisX.error,
                           errorID => "Unit1.Em7.ControlNodes".cm.calculateCam.sepaClampnCutterAxisX.errorID);
END_REGION

REGION Network 84: CmSepaClampnCutterAxisX SoftCam
   RUNG wire#powerrail
      "LER_SoftCam_Interface_FC"(actualPosition := "Unit1.Em7.HmiInterface".cmSepaClampnCutterAxisX.monitoring.actualPosition, selectSetPosition := "Unit1.Em7.HmiInterface".cmSepaClampnCutterAxisX.monitoring.selectSetPosition, softCam := "Unit1.Em7.Config".softCam.cmSepaClampnCutterAxisX, position := "Unit1.Em7.Config".cmSepaClampnCutterAxisX.setPositions, range := 0.01, softCamPos => "Unit1.Em7.ControlNodes".cm.softCam.sepaClampnCutterAxisX)
   END_RUNG
   // the same network as SCL:
   "LER_SoftCam_Interface_FC"(actualPosition := "Unit1.Em7.HmiInterface".cmSepaClampnCutterAxisX.monitoring.actualPosition,
                           selectSetPosition := "Unit1.Em7.HmiInterface".cmSepaClampnCutterAxisX.monitoring.selectSetPosition,
                           softCam := "Unit1.Em7.Config".softCam.cmSepaClampnCutterAxisX,
                           position := "Unit1.Em7.Config".cmSepaClampnCutterAxisX.setPositions,
                           range := 0.01,
                           softCamPos => "Unit1.Em7.ControlNodes".cm.softCam.sepaClampnCutterAxisX);
END_REGION

REGION Network 86: SepaClampnCutterAxisZ Enable
   RUNG wire#powerrail
      Contact( "Unit1.EmNodes".sleep.command.Servo.sleep )
      wire#w1
      R_Coil( "Unit1.Em7.ControlNodes".cmSepaClampnCutterAxisZ.commands.enableAxis )
   END_RUNG
   RUNG wire#powerrail
      Contact( "Unit1.EmNodes".sleep.command.Servo.deppSleep )
   END_RUNG wire#w1
   RUNG wire#powerrail
      Contact( "Unit1.EmNodes".sleep.State.WakeupRecovery )
      S_Coil( "Unit1.Em7.ControlNodes".cmSepaClampnCutterAxisZ.commands.enableAxis )
   END_RUNG
   // the same network as SCL:
   IF "Unit1.EmNodes".sleep.command.Servo.sleep OR "Unit1.EmNodes".sleep.command.Servo.deppSleep THEN
       "Unit1.Em7.ControlNodes".cmSepaClampnCutterAxisZ.commands.enableAxis := FALSE;
   END_IF;
   IF "Unit1.EmNodes".sleep.State.WakeupRecovery THEN
       "Unit1.Em7.ControlNodes".cmSepaClampnCutterAxisZ.commands.enableAxis := TRUE;
   END_IF;
END_REGION

REGION Network 87: CmSepaClampnCutterAxisZ Position Absolute Home
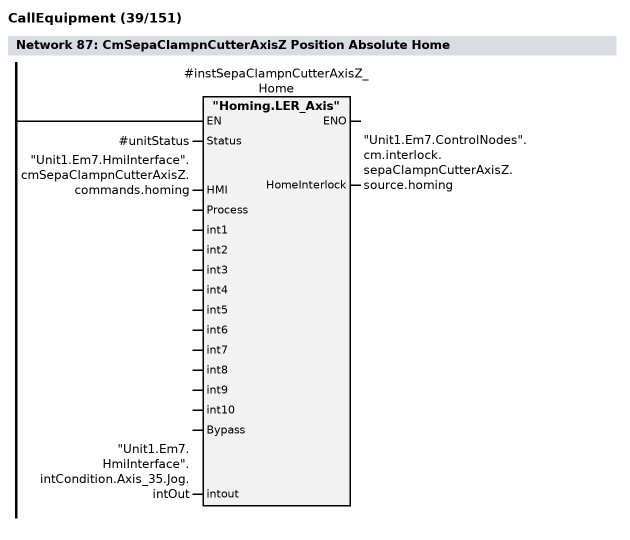
   RUNG wire#powerrail
      #instSepaClampnCutterAxisZ_Home(Status := #unitStatus, HMI := "Unit1.Em7.HmiInterface".cmSepaClampnCutterAxisZ.commands.homing, Process :=, int1 :=, int2 :=, int3 :=, int4 :=, int5 :=, int6 :=, int7 :=, int8 :=, int9 :=, int10 :=, Bypass :=, intout := "Unit1.Em7.HmiInterface".intCondition.Axis_35.Jog.intOut, HomeInterlock => "Unit1.Em7.ControlNodes".cm.interlock.sepaClampnCutterAxisZ.source.homing)
   END_RUNG
   // the same network as SCL:
   #instSepaClampnCutterAxisZ_Home(Status := #unitStatus,   // "Homing.LER_Axis"
                           HMI := "Unit1.Em7.HmiInterface".cmSepaClampnCutterAxisZ.commands.homing,
                           intout := "Unit1.Em7.HmiInterface".intCondition.Axis_35.Jog.intOut,
                           HomeInterlock => "Unit1.Em7.ControlNodes".cm.interlock.sepaClampnCutterAxisZ.source.homing);
END_REGION

REGION Network 88: CmSepaClampnCutterAxisZ Position Absolute Jog
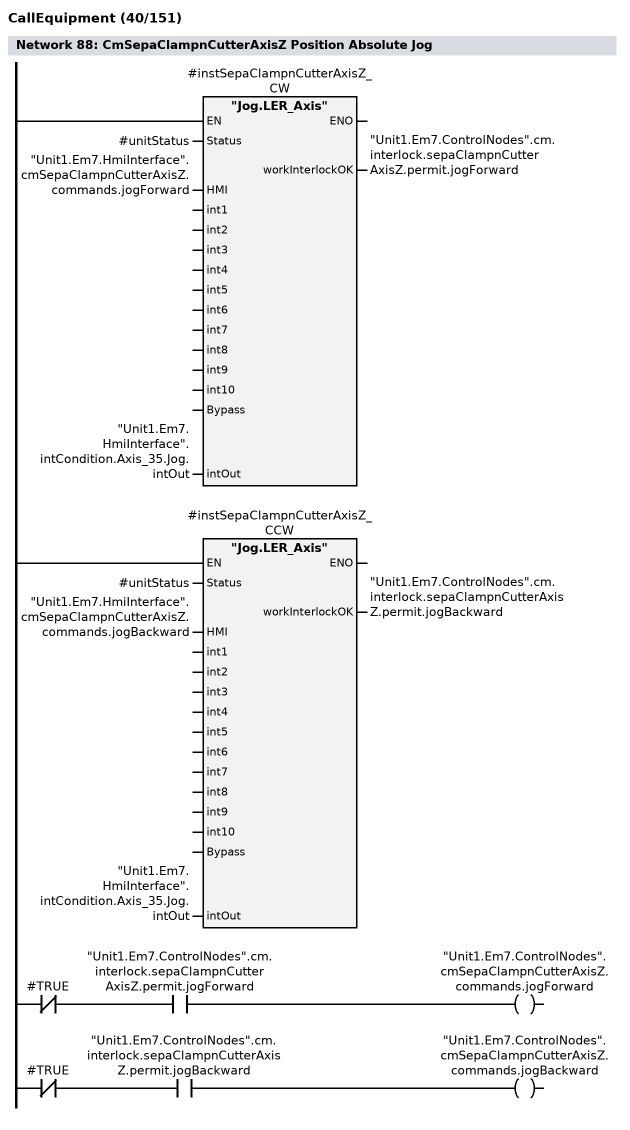
   RUNG wire#powerrail
      #instSepaClampnCutterAxisZ_CW(Status := #unitStatus, HMI := "Unit1.Em7.HmiInterface".cmSepaClampnCutterAxisZ.commands.jogForward, int1 :=, int2 :=, int3 :=, int4 :=, int5 :=, int6 :=, int7 :=, int8 :=, int9 :=, int10 :=, Bypass :=, intOut := "Unit1.Em7.HmiInterface".intCondition.Axis_35.Jog.intOut, workInterlockOK => "Unit1.Em7.ControlNodes".cm.interlock.sepaClampnCutterAxisZ.permit.jogForward)
   END_RUNG
   RUNG wire#powerrail
      #instSepaClampnCutterAxisZ_CCW(Status := #unitStatus, HMI := "Unit1.Em7.HmiInterface".cmSepaClampnCutterAxisZ.commands.jogBackward, int1 :=, int2 :=, int3 :=, int4 :=, int5 :=, int6 :=, int7 :=, int8 :=, int9 :=, int10 :=, Bypass :=, intOut := "Unit1.Em7.HmiInterface".intCondition.Axis_35.Jog.intOut, workInterlockOK => "Unit1.Em7.ControlNodes".cm.interlock.sepaClampnCutterAxisZ.permit.jogBackward)
   END_RUNG
   RUNG wire#powerrail
      I_Contact( #TRUE )
      Contact( "Unit1.Em7.ControlNodes".cm.interlock.sepaClampnCutterAxisZ.permit.jogForward )
      Coil( "Unit1.Em7.ControlNodes".cmSepaClampnCutterAxisZ.commands.jogForward )
   END_RUNG
   RUNG wire#powerrail
      I_Contact( #TRUE )
      Contact( "Unit1.Em7.ControlNodes".cm.interlock.sepaClampnCutterAxisZ.permit.jogBackward )
      Coil( "Unit1.Em7.ControlNodes".cmSepaClampnCutterAxisZ.commands.jogBackward )
   END_RUNG
   // the same network as SCL:
   #instSepaClampnCutterAxisZ_CW(Status := #unitStatus,   // "Jog.LER_Axis"
                           HMI := "Unit1.Em7.HmiInterface".cmSepaClampnCutterAxisZ.commands.jogForward,
                           intOut := "Unit1.Em7.HmiInterface".intCondition.Axis_35.Jog.intOut,
                           workInterlockOK => "Unit1.Em7.ControlNodes".cm.interlock.sepaClampnCutterAxisZ.permit.jogForward);
   #instSepaClampnCutterAxisZ_CCW(Status := #unitStatus,   // "Jog.LER_Axis"
                           HMI := "Unit1.Em7.HmiInterface".cmSepaClampnCutterAxisZ.commands.jogBackward,
                           intOut := "Unit1.Em7.HmiInterface".intCondition.Axis_35.Jog.intOut,
                           workInterlockOK => "Unit1.Em7.ControlNodes".cm.interlock.sepaClampnCutterAxisZ.permit.jogBackward);
   "Unit1.Em7.ControlNodes".cmSepaClampnCutterAxisZ.commands.jogForward := NOT #TRUE AND "Unit1.Em7.ControlNodes".cm.interlock.sepaClampnCutterAxisZ.permit.jogForward;
   "Unit1.Em7.ControlNodes".cmSepaClampnCutterAxisZ.commands.jogBackward := NOT #TRUE AND "Unit1.Em7.ControlNodes".cm.interlock.sepaClampnCutterAxisZ.permit.jogBackward;
END_REGION

REGION Network 89: CmSepaClampnCutterAxisZ Position Absolute Position0
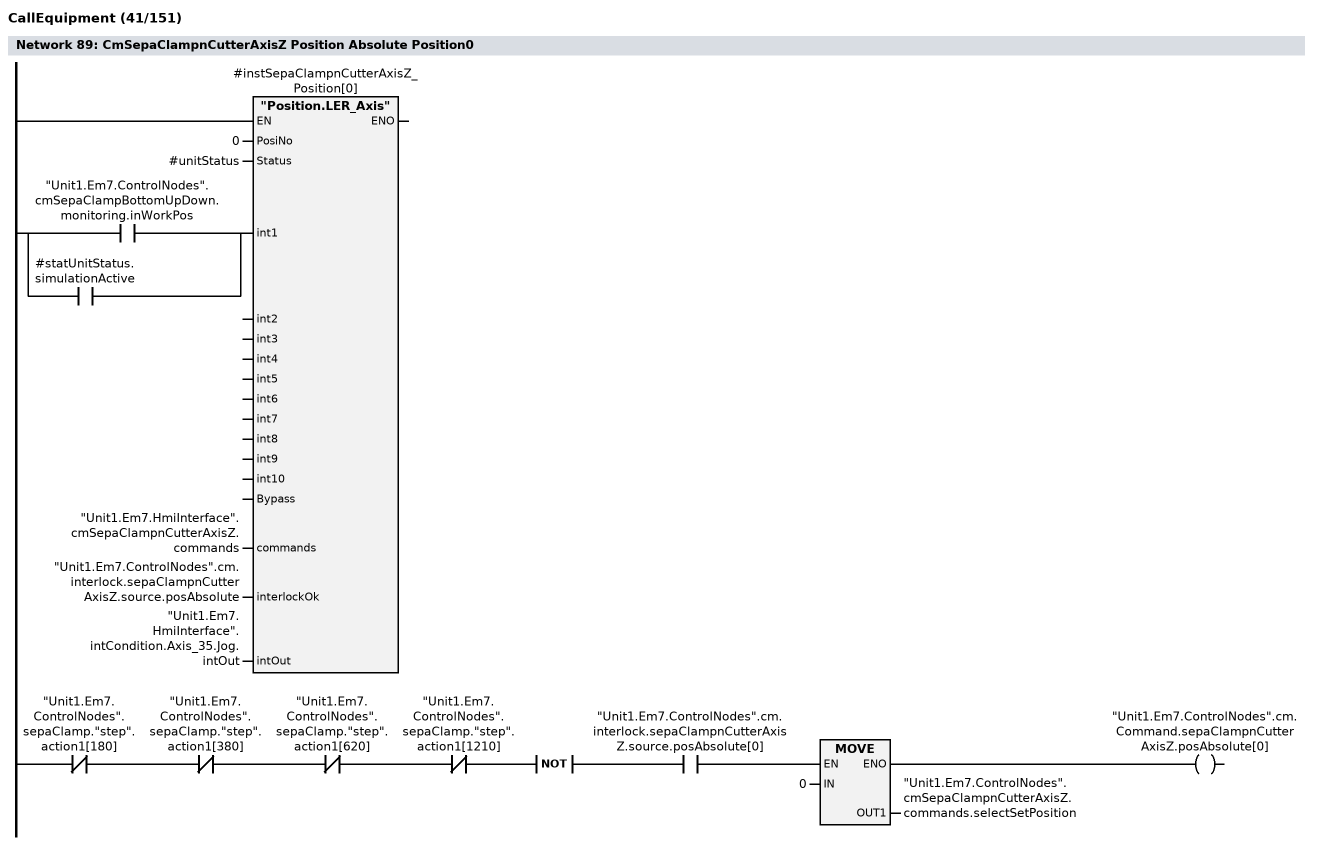
   RUNG wire#powerrail
      #instSepaClampnCutterAxisZ_Position[0](int1 := wire#w1, PosiNo := 0, Status := #unitStatus, int2 :=, int3 :=, int4 :=, int5 :=, int6 :=, int7 :=, int8 :=, int9 :=, int10 :=, Bypass :=, commands := "Unit1.Em7.HmiInterface".cmSepaClampnCutterAxisZ.commands, interlockOk := "Unit1.Em7.ControlNodes".cm.interlock.sepaClampnCutterAxisZ.source.posAbsolute, intOut := "Unit1.Em7.HmiInterface".intCondition.Axis_35.Jog.intOut)
   END_RUNG
   RUNG wire#powerrail
      Contact( "Unit1.Em7.ControlNodes".cmSepaClampBottomUpDown.monitoring.inWorkPos )
   END_RUNG wire#w1
   RUNG wire#powerrail
      Contact( #statUnitStatus.simulationActive )
   END_RUNG wire#w1
   RUNG wire#powerrail
      I_Contact( "Unit1.Em7.ControlNodes".sepaClamp."step".action1[180] )
      I_Contact( "Unit1.Em7.ControlNodes".sepaClamp."step".action1[380] )
      I_Contact( "Unit1.Em7.ControlNodes".sepaClamp."step".action1[620] )
      I_Contact( "Unit1.Em7.ControlNodes".sepaClamp."step".action1[1210] )
      Not()
      Contact( "Unit1.Em7.ControlNodes".cm.interlock.sepaClampnCutterAxisZ.source.posAbsolute[0] )
      Move(in := 0, out1 => "Unit1.Em7.ControlNodes".cmSepaClampnCutterAxisZ.commands.selectSetPosition)
      Coil( "Unit1.Em7.ControlNodes".cm.Command.sepaClampnCutterAxisZ.posAbsolute[0] )
   END_RUNG
   // the same network as SCL:
   #instSepaClampnCutterAxisZ_Position[0](PosiNo := 0,   // "Position.LER_Axis"
                           Status := #unitStatus,
                           int1 := "Unit1.Em7.ControlNodes".cmSepaClampBottomUpDown.monitoring.inWorkPos OR #statUnitStatus.simulationActive,
                           commands := "Unit1.Em7.HmiInterface".cmSepaClampnCutterAxisZ.commands,
                           interlockOk := "Unit1.Em7.ControlNodes".cm.interlock.sepaClampnCutterAxisZ.source.posAbsolute,
                           intOut := "Unit1.Em7.HmiInterface".intCondition.Axis_35.Jog.intOut);
   #_w1 := NOT (NOT "Unit1.Em7.ControlNodes".sepaClamp."step".action1[180] AND NOT "Unit1.Em7.ControlNodes".sepaClamp."step".action1[380] AND NOT "Unit1.Em7.ControlNodes".sepaClamp."step".action1[620] AND NOT "Unit1.Em7.ControlNodes".sepaClamp."step".action1[1210]) AND "Unit1.Em7.ControlNodes".cm.interlock.sepaClampnCutterAxisZ.source.posAbsolute[0];
   IF #_w1 THEN "Unit1.Em7.ControlNodes".cmSepaClampnCutterAxisZ.commands.selectSetPosition := 0; END_IF;
   "Unit1.Em7.ControlNodes".cm.Command.sepaClampnCutterAxisZ.posAbsolute[0] := #_w1;
END_REGION

REGION Network 90: CmSepaClampnCutterAxisZ Position Absolute Position1
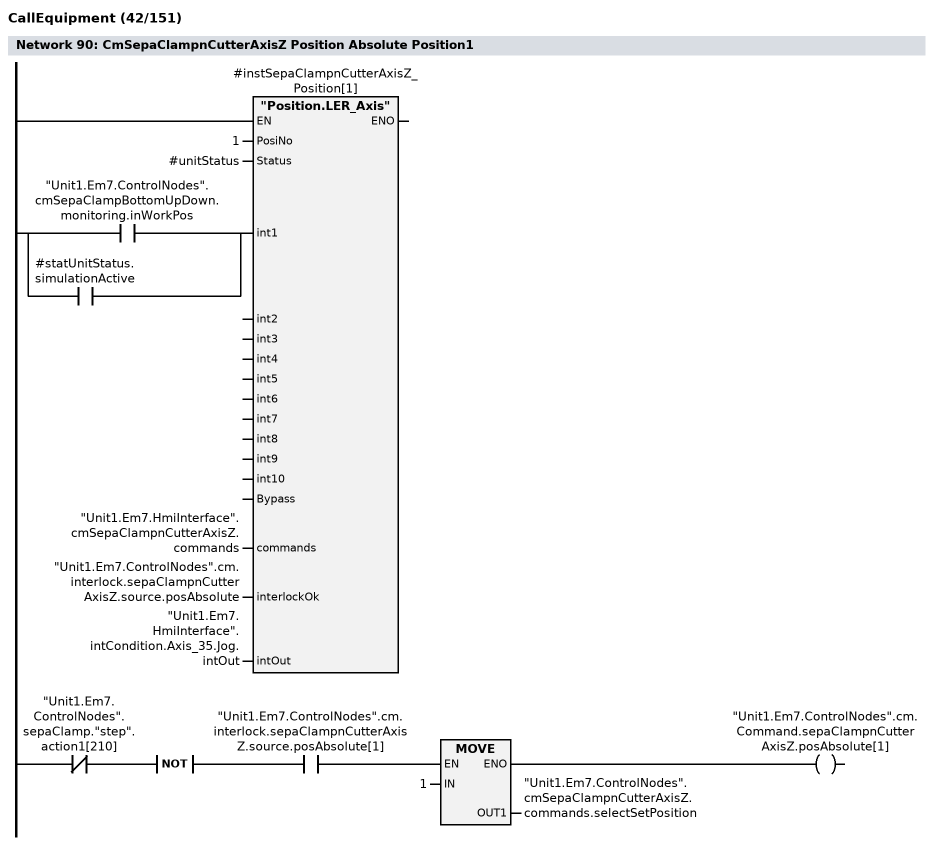
   RUNG wire#powerrail
      #instSepaClampnCutterAxisZ_Position[1](int1 := wire#w1, PosiNo := 1, Status := #unitStatus, int2 :=, int3 :=, int4 :=, int5 :=, int6 :=, int7 :=, int8 :=, int9 :=, int10 :=, Bypass :=, commands := "Unit1.Em7.HmiInterface".cmSepaClampnCutterAxisZ.commands, interlockOk := "Unit1.Em7.ControlNodes".cm.interlock.sepaClampnCutterAxisZ.source.posAbsolute, intOut := "Unit1.Em7.HmiInterface".intCondition.Axis_35.Jog.intOut)
   END_RUNG
   RUNG wire#powerrail
      Contact( "Unit1.Em7.ControlNodes".cmSepaClampBottomUpDown.monitoring.inWorkPos )
   END_RUNG wire#w1
   RUNG wire#powerrail
      Contact( #statUnitStatus.simulationActive )
   END_RUNG wire#w1
   RUNG wire#powerrail
      I_Contact( "Unit1.Em7.ControlNodes".sepaClamp."step".action1[210] )
      Not()
      Contact( "Unit1.Em7.ControlNodes".cm.interlock.sepaClampnCutterAxisZ.source.posAbsolute[1] )
      Move(in := 1, out1 => "Unit1.Em7.ControlNodes".cmSepaClampnCutterAxisZ.commands.selectSetPosition)
      Coil( "Unit1.Em7.ControlNodes".cm.Command.sepaClampnCutterAxisZ.posAbsolute[1] )
   END_RUNG
   // the same network as SCL:
   #instSepaClampnCutterAxisZ_Position[1](PosiNo := 1,   // "Position.LER_Axis"
                           Status := #unitStatus,
                           int1 := "Unit1.Em7.ControlNodes".cmSepaClampBottomUpDown.monitoring.inWorkPos OR #statUnitStatus.simulationActive,
                           commands := "Unit1.Em7.HmiInterface".cmSepaClampnCutterAxisZ.commands,
                           interlockOk := "Unit1.Em7.ControlNodes".cm.interlock.sepaClampnCutterAxisZ.source.posAbsolute,
                           intOut := "Unit1.Em7.HmiInterface".intCondition.Axis_35.Jog.intOut);
   #_w1 := NOT (NOT "Unit1.Em7.ControlNodes".sepaClamp."step".action1[210]) AND "Unit1.Em7.ControlNodes".cm.interlock.sepaClampnCutterAxisZ.source.posAbsolute[1];
   IF #_w1 THEN "Unit1.Em7.ControlNodes".cmSepaClampnCutterAxisZ.commands.selectSetPosition := 1; END_IF;
   "Unit1.Em7.ControlNodes".cm.Command.sepaClampnCutterAxisZ.posAbsolute[1] := #_w1;
END_REGION

REGION Network 91: CmSepaClampnCutterAxisZ Position Absolute Position2
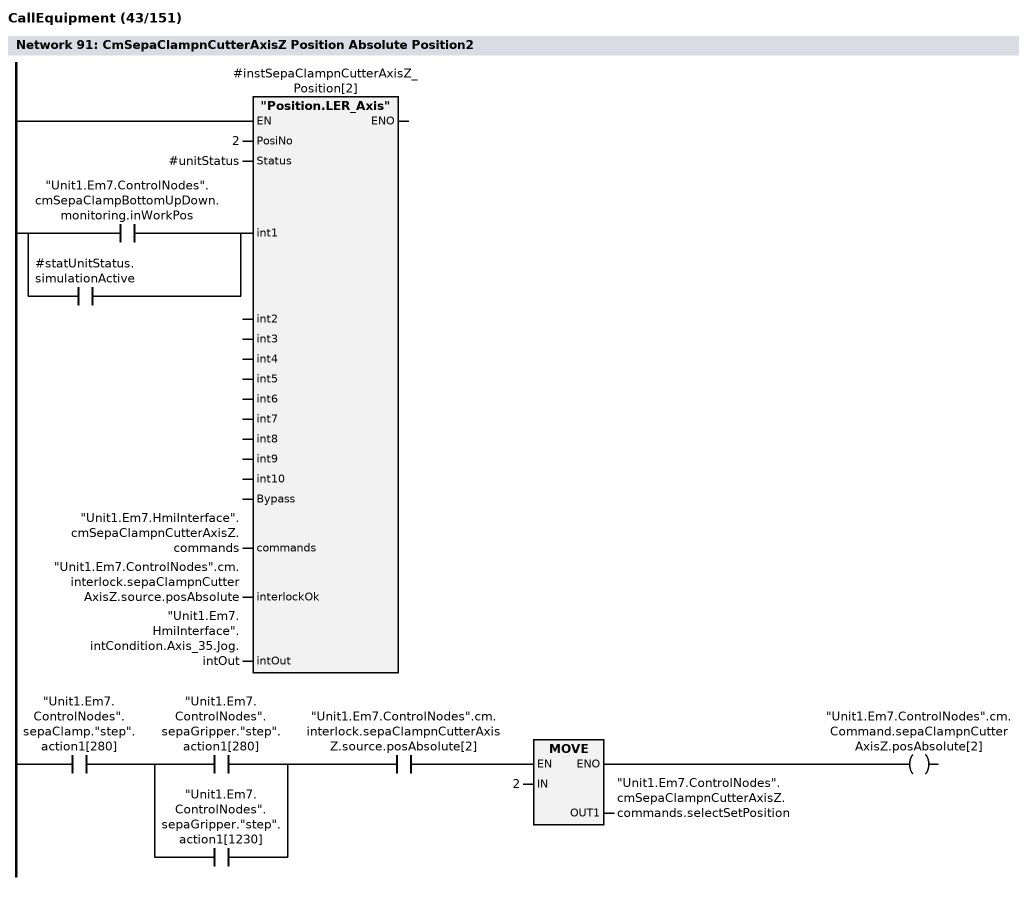
   RUNG wire#powerrail
      #instSepaClampnCutterAxisZ_Position[2](int1 := wire#w1, PosiNo := 2, Status := #unitStatus, int2 :=, int3 :=, int4 :=, int5 :=, int6 :=, int7 :=, int8 :=, int9 :=, int10 :=, Bypass :=, commands := "Unit1.Em7.HmiInterface".cmSepaClampnCutterAxisZ.commands, interlockOk := "Unit1.Em7.ControlNodes".cm.interlock.sepaClampnCutterAxisZ.source.posAbsolute, intOut := "Unit1.Em7.HmiInterface".intCondition.Axis_35.Jog.intOut)
   END_RUNG
   RUNG wire#powerrail
      Contact( "Unit1.Em7.ControlNodes".cmSepaClampBottomUpDown.monitoring.inWorkPos )
   END_RUNG wire#w1
   RUNG wire#powerrail
      Contact( #statUnitStatus.simulationActive )
   END_RUNG wire#w1
   RUNG wire#powerrail
      Contact( "Unit1.Em7.ControlNodes".sepaClamp."step".action1[280] )
      wire#w2
      Contact( "Unit1.Em7.ControlNodes".sepaGripper."step".action1[280] )
      wire#w3
      Contact( "Unit1.Em7.ControlNodes".cm.interlock.sepaClampnCutterAxisZ.source.posAbsolute[2] )
      Move(in := 2, out1 => "Unit1.Em7.ControlNodes".cmSepaClampnCutterAxisZ.commands.selectSetPosition)
      Coil( "Unit1.Em7.ControlNodes".cm.Command.sepaClampnCutterAxisZ.posAbsolute[2] )
   END_RUNG
   RUNG wire#w2
      Contact( "Unit1.Em7.ControlNodes".sepaGripper."step".action1[1230] )
   END_RUNG wire#w3
   // the same network as SCL:
   #instSepaClampnCutterAxisZ_Position[2](PosiNo := 2,   // "Position.LER_Axis"
                           Status := #unitStatus,
                           int1 := "Unit1.Em7.ControlNodes".cmSepaClampBottomUpDown.monitoring.inWorkPos OR #statUnitStatus.simulationActive,
                           commands := "Unit1.Em7.HmiInterface".cmSepaClampnCutterAxisZ.commands,
                           interlockOk := "Unit1.Em7.ControlNodes".cm.interlock.sepaClampnCutterAxisZ.source.posAbsolute,
                           intOut := "Unit1.Em7.HmiInterface".intCondition.Axis_35.Jog.intOut);
   #_w1 := "Unit1.Em7.ControlNodes".sepaClamp."step".action1[280] AND ("Unit1.Em7.ControlNodes".sepaGripper."step".action1[280] OR "Unit1.Em7.ControlNodes".sepaGripper."step".action1[1230]) AND "Unit1.Em7.ControlNodes".cm.interlock.sepaClampnCutterAxisZ.source.posAbsolute[2];
   IF #_w1 THEN "Unit1.Em7.ControlNodes".cmSepaClampnCutterAxisZ.commands.selectSetPosition := 2; END_IF;
   "Unit1.Em7.ControlNodes".cm.Command.sepaClampnCutterAxisZ.posAbsolute[2] := #_w1;
END_REGION

REGION Network 92: CmSepaClampnCutterAxisZ Position Absolute Position3
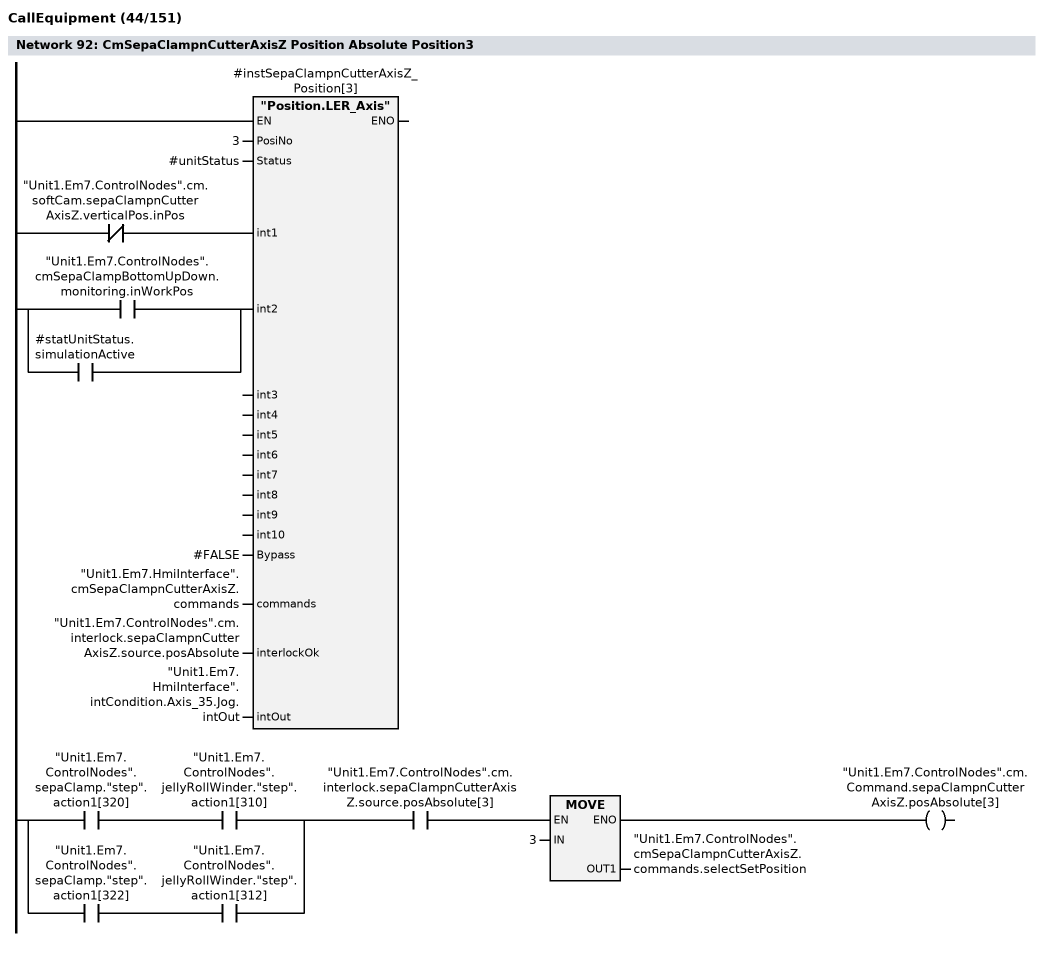
   RUNG wire#powerrail
      #instSepaClampnCutterAxisZ_Position[3](int1 := wire#w1, int2 := wire#w2, PosiNo := 3, Status := #unitStatus, int3 :=, int4 :=, int5 :=, int6 :=, int7 :=, int8 :=, int9 :=, int10 :=, Bypass := #FALSE, commands := "Unit1.Em7.HmiInterface".cmSepaClampnCutterAxisZ.commands, interlockOk := "Unit1.Em7.ControlNodes".cm.interlock.sepaClampnCutterAxisZ.source.posAbsolute, intOut := "Unit1.Em7.HmiInterface".intCondition.Axis_35.Jog.intOut)
   END_RUNG
   RUNG wire#powerrail
      I_Contact( "Unit1.Em7.ControlNodes".cm.softCam.sepaClampnCutterAxisZ.verticalPos.inPos )
   END_RUNG wire#w1
   RUNG wire#powerrail
      Contact( "Unit1.Em7.ControlNodes".cmSepaClampBottomUpDown.monitoring.inWorkPos )
   END_RUNG wire#w2
   RUNG wire#powerrail
      Contact( #statUnitStatus.simulationActive )
   END_RUNG wire#w2
   RUNG wire#powerrail
      Contact( "Unit1.Em7.ControlNodes".sepaClamp."step".action1[320] )
      Contact( "Unit1.Em7.ControlNodes".jellyRollWinder."step".action1[310] )
      wire#w3
      Contact( "Unit1.Em7.ControlNodes".cm.interlock.sepaClampnCutterAxisZ.source.posAbsolute[3] )
      Move(in := 3, out1 => "Unit1.Em7.ControlNodes".cmSepaClampnCutterAxisZ.commands.selectSetPosition)
      Coil( "Unit1.Em7.ControlNodes".cm.Command.sepaClampnCutterAxisZ.posAbsolute[3] )
   END_RUNG
   RUNG wire#powerrail
      Contact( "Unit1.Em7.ControlNodes".sepaClamp."step".action1[322] )
      Contact( "Unit1.Em7.ControlNodes".jellyRollWinder."step".action1[312] )
   END_RUNG wire#w3
   // the same network as SCL:
   #instSepaClampnCutterAxisZ_Position[3](PosiNo := 3,   // "Position.LER_Axis"
                           Status := #unitStatus,
                           int1 := NOT "Unit1.Em7.ControlNodes".cm.softCam.sepaClampnCutterAxisZ.verticalPos.inPos,
                           int2 := "Unit1.Em7.ControlNodes".cmSepaClampBottomUpDown.monitoring.inWorkPos OR #statUnitStatus.simulationActive,
                           Bypass := #FALSE,
                           commands := "Unit1.Em7.HmiInterface".cmSepaClampnCutterAxisZ.commands,
                           interlockOk := "Unit1.Em7.ControlNodes".cm.interlock.sepaClampnCutterAxisZ.source.posAbsolute,
                           intOut := "Unit1.Em7.HmiInterface".intCondition.Axis_35.Jog.intOut);
   #_w1 := (("Unit1.Em7.ControlNodes".sepaClamp."step".action1[320] AND "Unit1.Em7.ControlNodes".jellyRollWinder."step".action1[310]) OR ("Unit1.Em7.ControlNodes".sepaClamp."step".action1[322] AND "Unit1.Em7.ControlNodes".jellyRollWinder."step".action1[312])) AND "Unit1.Em7.ControlNodes".cm.interlock.sepaClampnCutterAxisZ.source.posAbsolute[3];
   IF #_w1 THEN "Unit1.Em7.ControlNodes".cmSepaClampnCutterAxisZ.commands.selectSetPosition := 3; END_IF;
   "Unit1.Em7.ControlNodes".cm.Command.sepaClampnCutterAxisZ.posAbsolute[3] := #_w1;
END_REGION

REGION Network 93: CmSepaClampnCutterAxisZ Position Absolute Position4
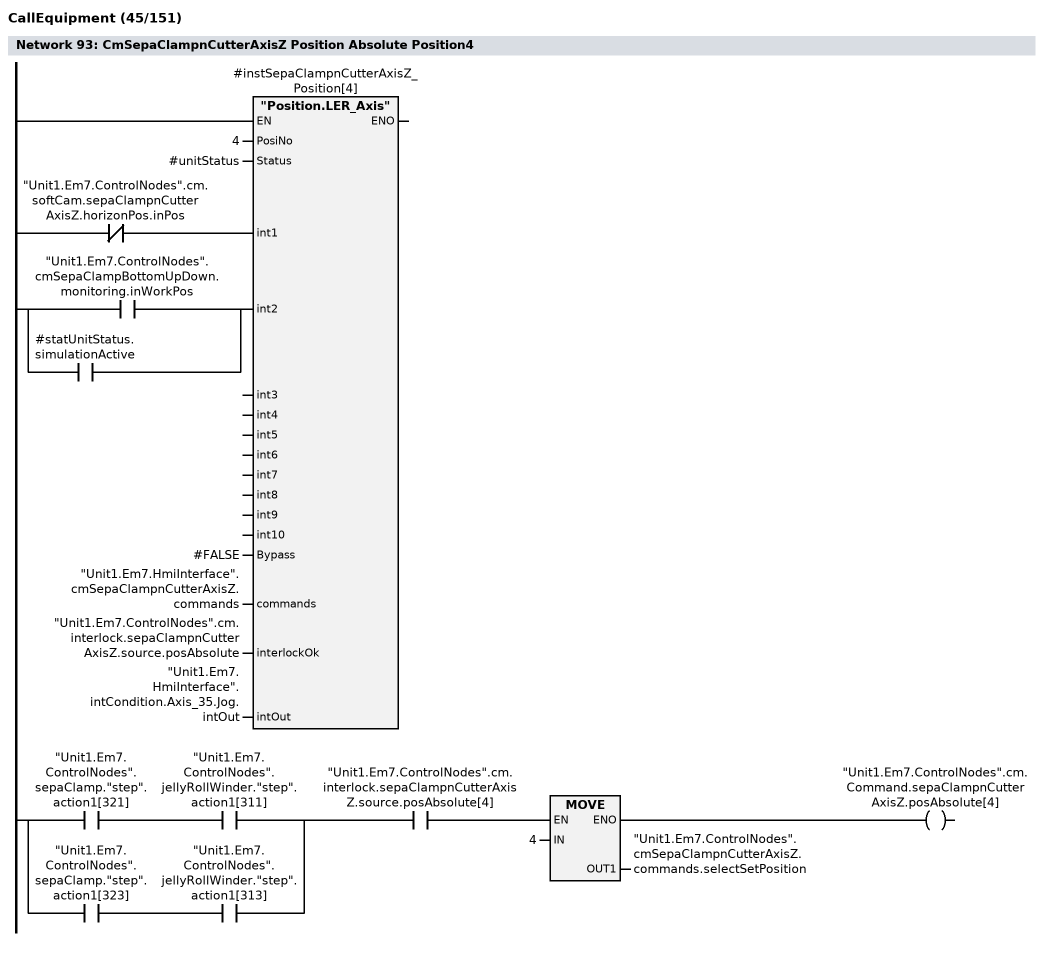
   RUNG wire#powerrail
      #instSepaClampnCutterAxisZ_Position[4](int1 := wire#w1, int2 := wire#w2, PosiNo := 4, Status := #unitStatus, int3 :=, int4 :=, int5 :=, int6 :=, int7 :=, int8 :=, int9 :=, int10 :=, Bypass := #FALSE, commands := "Unit1.Em7.HmiInterface".cmSepaClampnCutterAxisZ.commands, interlockOk := "Unit1.Em7.ControlNodes".cm.interlock.sepaClampnCutterAxisZ.source.posAbsolute, intOut := "Unit1.Em7.HmiInterface".intCondition.Axis_35.Jog.intOut)
   END_RUNG
   RUNG wire#powerrail
      I_Contact( "Unit1.Em7.ControlNodes".cm.softCam.sepaClampnCutterAxisZ.horizonPos.inPos )
   END_RUNG wire#w1
   RUNG wire#powerrail
      Contact( "Unit1.Em7.ControlNodes".cmSepaClampBottomUpDown.monitoring.inWorkPos )
   END_RUNG wire#w2
   RUNG wire#powerrail
      Contact( #statUnitStatus.simulationActive )
   END_RUNG wire#w2
   RUNG wire#powerrail
      Contact( "Unit1.Em7.ControlNodes".sepaClamp."step".action1[321] )
      Contact( "Unit1.Em7.ControlNodes".jellyRollWinder."step".action1[311] )
      wire#w3
      Contact( "Unit1.Em7.ControlNodes".cm.interlock.sepaClampnCutterAxisZ.source.posAbsolute[4] )
      Move(in := 4, out1 => "Unit1.Em7.ControlNodes".cmSepaClampnCutterAxisZ.commands.selectSetPosition)
      Coil( "Unit1.Em7.ControlNodes".cm.Command.sepaClampnCutterAxisZ.posAbsolute[4] )
   END_RUNG
   RUNG wire#powerrail
      Contact( "Unit1.Em7.ControlNodes".sepaClamp."step".action1[323] )
      Contact( "Unit1.Em7.ControlNodes".jellyRollWinder."step".action1[313] )
   END_RUNG wire#w3
   // the same network as SCL:
   #instSepaClampnCutterAxisZ_Position[4](PosiNo := 4,   // "Position.LER_Axis"
                           Status := #unitStatus,
                           int1 := NOT "Unit1.Em7.ControlNodes".cm.softCam.sepaClampnCutterAxisZ.horizonPos.inPos,
                           int2 := "Unit1.Em7.ControlNodes".cmSepaClampBottomUpDown.monitoring.inWorkPos OR #statUnitStatus.simulationActive,
                           Bypass := #FALSE,
                           commands := "Unit1.Em7.HmiInterface".cmSepaClampnCutterAxisZ.commands,
                           interlockOk := "Unit1.Em7.ControlNodes".cm.interlock.sepaClampnCutterAxisZ.source.posAbsolute,
                           intOut := "Unit1.Em7.HmiInterface".intCondition.Axis_35.Jog.intOut);
   #_w1 := (("Unit1.Em7.ControlNodes".sepaClamp."step".action1[321] AND "Unit1.Em7.ControlNodes".jellyRollWinder."step".action1[311]) OR ("Unit1.Em7.ControlNodes".sepaClamp."step".action1[323] AND "Unit1.Em7.ControlNodes".jellyRollWinder."step".action1[313])) AND "Unit1.Em7.ControlNodes".cm.interlock.sepaClampnCutterAxisZ.source.posAbsolute[4];
   IF #_w1 THEN "Unit1.Em7.ControlNodes".cmSepaClampnCutterAxisZ.commands.selectSetPosition := 4; END_IF;
   "Unit1.Em7.ControlNodes".cm.Command.sepaClampnCutterAxisZ.posAbsolute[4] := #_w1;
END_REGION

REGION Network 94: CmSepaClampnCutterAxisZ Position Absolute Position5
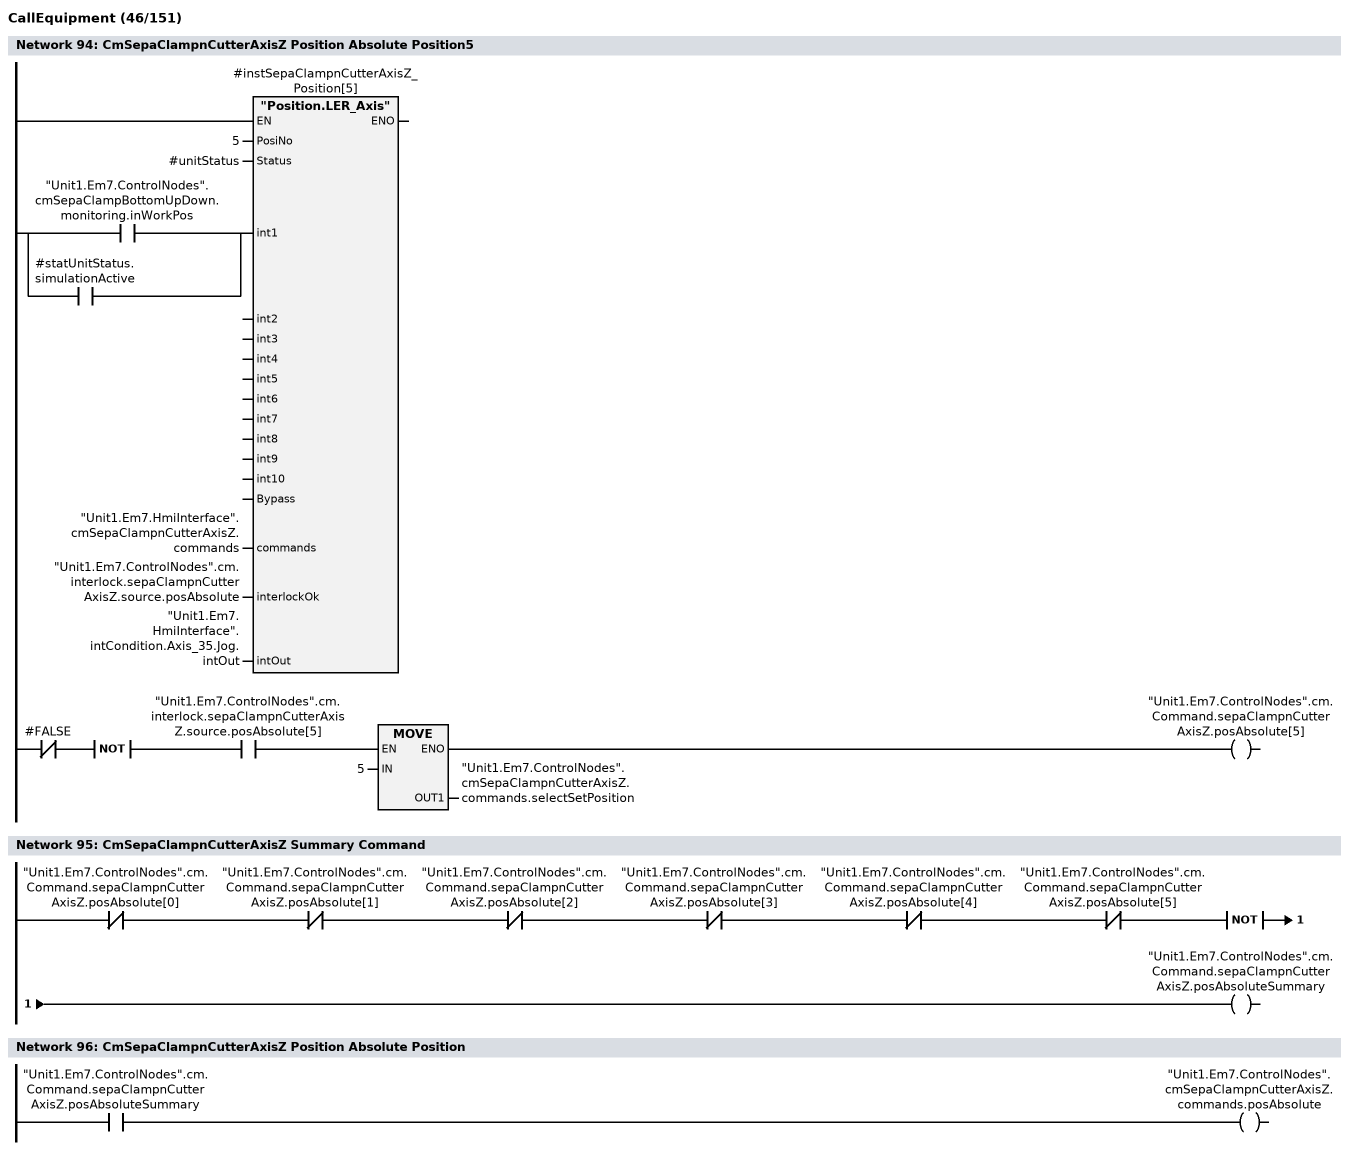
   RUNG wire#powerrail
      #instSepaClampnCutterAxisZ_Position[5](int1 := wire#w1, PosiNo := 5, Status := #unitStatus, int2 :=, int3 :=, int4 :=, int5 :=, int6 :=, int7 :=, int8 :=, int9 :=, int10 :=, Bypass :=, commands := "Unit1.Em7.HmiInterface".cmSepaClampnCutterAxisZ.commands, interlockOk := "Unit1.Em7.ControlNodes".cm.interlock.sepaClampnCutterAxisZ.source.posAbsolute, intOut := "Unit1.Em7.HmiInterface".intCondition.Axis_35.Jog.intOut)
   END_RUNG
   RUNG wire#powerrail
      Contact( "Unit1.Em7.ControlNodes".cmSepaClampBottomUpDown.monitoring.inWorkPos )
   END_RUNG wire#w1
   RUNG wire#powerrail
      Contact( #statUnitStatus.simulationActive )
   END_RUNG wire#w1
   RUNG wire#powerrail
      I_Contact( #FALSE )
      Not()
      Contact( "Unit1.Em7.ControlNodes".cm.interlock.sepaClampnCutterAxisZ.source.posAbsolute[5] )
      Move(in := 5, out1 => "Unit1.Em7.ControlNodes".cmSepaClampnCutterAxisZ.commands.selectSetPosition)
      Coil( "Unit1.Em7.ControlNodes".cm.Command.sepaClampnCutterAxisZ.posAbsolute[5] )
   END_RUNG
   // the same network as SCL:
   #instSepaClampnCutterAxisZ_Position[5](PosiNo := 5,   // "Position.LER_Axis"
                           Status := #unitStatus,
                           int1 := "Unit1.Em7.ControlNodes".cmSepaClampBottomUpDown.monitoring.inWorkPos OR #statUnitStatus.simulationActive,
                           commands := "Unit1.Em7.HmiInterface".cmSepaClampnCutterAxisZ.commands,
                           interlockOk := "Unit1.Em7.ControlNodes".cm.interlock.sepaClampnCutterAxisZ.source.posAbsolute,
                           intOut := "Unit1.Em7.HmiInterface".intCondition.Axis_35.Jog.intOut);
   #_w1 := NOT (NOT #FALSE) AND "Unit1.Em7.ControlNodes".cm.interlock.sepaClampnCutterAxisZ.source.posAbsolute[5];
   IF #_w1 THEN "Unit1.Em7.ControlNodes".cmSepaClampnCutterAxisZ.commands.selectSetPosition := 5; END_IF;
   "Unit1.Em7.ControlNodes".cm.Command.sepaClampnCutterAxisZ.posAbsolute[5] := #_w1;
END_REGION

REGION Network 95: CmSepaClampnCutterAxisZ Summary Command
   RUNG wire#powerrail
      I_Contact( "Unit1.Em7.ControlNodes".cm.Command.sepaClampnCutterAxisZ.posAbsolute[0] )
      I_Contact( "Unit1.Em7.ControlNodes".cm.Command.sepaClampnCutterAxisZ.posAbsolute[1] )
      I_Contact( "Unit1.Em7.ControlNodes".cm.Command.sepaClampnCutterAxisZ.posAbsolute[2] )
      I_Contact( "Unit1.Em7.ControlNodes".cm.Command.sepaClampnCutterAxisZ.posAbsolute[3] )
      I_Contact( "Unit1.Em7.ControlNodes".cm.Command.sepaClampnCutterAxisZ.posAbsolute[4] )
      I_Contact( "Unit1.Em7.ControlNodes".cm.Command.sepaClampnCutterAxisZ.posAbsolute[5] )
      Not()
      Coil( "Unit1.Em7.ControlNodes".cm.Command.sepaClampnCutterAxisZ.posAbsoluteSummary )
   END_RUNG
   // the same network as SCL:
   "Unit1.Em7.ControlNodes".cm.Command.sepaClampnCutterAxisZ.posAbsoluteSummary := NOT (NOT "Unit1.Em7.ControlNodes".cm.Command.sepaClampnCutterAxisZ.posAbsolute[0] AND NOT "Unit1.Em7.ControlNodes".cm.Command.sepaClampnCutterAxisZ.posAbsolute[1] AND NOT "Unit1.Em7.ControlNodes".cm.Command.sepaClampnCutterAxisZ.posAbsolute[2] AND NOT "Unit1.Em7.ControlNodes".cm.Command.sepaClampnCutterAxisZ.posAbsolute[3] AND NOT "Unit1.Em7.ControlNodes".cm.Command.sepaClampnCutterAxisZ.posAbsolute[4] AND NOT "Unit1.Em7.ControlNodes".cm.Command.sepaClampnCutterAxisZ.posAbsolute[5]);
END_REGION

REGION Network 96: CmSepaClampnCutterAxisZ Position Absolute Position
   RUNG wire#powerrail
      Contact( "Unit1.Em7.ControlNodes".cm.Command.sepaClampnCutterAxisZ.posAbsoluteSummary )
      Coil( "Unit1.Em7.ControlNodes".cmSepaClampnCutterAxisZ.commands.posAbsolute )
   END_RUNG
   // the same network as SCL:
   "Unit1.Em7.ControlNodes".cmSepaClampnCutterAxisZ.commands.posAbsolute := "Unit1.Em7.ControlNodes".cm.Command.sepaClampnCutterAxisZ.posAbsoluteSummary;
END_REGION

REGION Network 97: CmSepaClampnCutterAxisZ Interlock Summary
